(* IEC 61131-3 sources: MIRA/plc (part 4) *)

(* ---- Micro820_v4.2.2_Program.st ---- *)
PROGRAM Prog2
(* ================================================================ *)
(*  MIRA Conveyor Control -- Micro820 2080-LC20-20QBB               *)
(*  Version:  v4.2.2                                                *)
(*  Date:     2026-06-27                                            *)
(*  Author:   MIRA/Codex                                            *)
(*                                                                  *)
(*  v4.2.2 is a bench/demo logic update on top of v4.1.9. It adds   *)
(*  supervised SimLab discharge request handling for the garage      *)
(*  conveyor when used as bottling-line discharge_conveyor01. This  *)
(*  is not production-certified machinery control. The real         *)
(*  Micro820/GS10 bench still owns motion and safety authority.     *)
(*                                                                  *)
(*  Changelog vs v4.1.9:                                            *)
(*   0. FIX v4.2.2 -- remove the extra safety-ok global requirement. *)
(*      CCW build proved that variable was not in the v4.2.0 delta.  *)
(*      Use existing e_stop_active / estop_wiring_fault directly.    *)
(*   1. NEW -- simlab_discharge_request is request-only. It never   *)
(*      writes directly to the VFD, motor, contactor, or outputs.   *)
(*   2. NEW -- discharge_pending_acceptance requires a local human  *)
(*      acceptance rising edge from PBRun / _IO_EM_DI_04.           *)
(*   3. NEW -- discharge_accept_timer rejects pending requests      *)
(*      after 30 seconds if no local acceptance arrives.             *)
(*   4. NEW -- photoeye_clear_timer requires DI05/photoeye clear    *)
(*      for 30 seconds before the next accepted discharge can run.  *)
(*   5. NEW -- accepted discharge stops when photoeye_blocked goes  *)
(*      TRUE, or on E-stop, stop/selector-off, drive comm fault,    *)
(*      active fault, heartbeat loss, request drop, or shutdown.    *)
(*   6. NEW -- amber_led_flash now drives the bench amber lamp on   *)
(*      O-04 / _IO_EM_DO_04 while discharge acceptance is pending.  *)
(*      Do not reuse DO0/DO1/DO2/DO3.                               *)
(*                                                                  *)
(*  Still deliberately deferred beyond v4.2.2:                      *)
(*   - Removal of vfd_cmd_word := N assignments throughout the      *)
(*     state machine. The TODO calls for the motor_starter UDFB     *)
(*     in Prog4 to become the sole writer. Until Prog4 ships,       *)
(*     removing these writes here would leave nothing commanding    *)
(*     the drive. Two writers in one scan is bad, zero writers      *)
(*     is worse. Will rip them out atomically with the Prog4 add.   *)
(*   - mb_read_status -> mb_read_monitor rename. That's a CCW       *)
(*     IDE instance rename + cross-reference cleanup. Not safe to   *)
(*     do via ST edit alone; do it in CCW. Comments below use the   *)
(*     accurate name (mb_read_monitor) so the rename is obvious.    *)
(*   - Poll timer 500ms -> 50ms tuning. Cosmetic right now; first   *)
(*     prove comms work, then tune.                                 *)
(*                                                                  *)
(*  NEW VARIABLES to declare in CCW Controller Variables table      *)
(*  (PrjLibrary.accdb -- DO NOT add a VAR block here):              *)
(*                                                                  *)
(*    Name                          Type                  Init      *)
(*    ----                          ----                  ----      *)
(*    commissioning_mode            BOOL                  (none)    *)
(*    read_status_word_local_cfg    MSGMODBUSPARA_LOCAL   (none)    *)
(*    read_status_word_target_cfg   MSGMODBUSPARA_TARGET  (none)    *)
(*    read_status_word_data         MODBUSLOCADDR[1..1]   (none)    *)
(*    mb_read_status_word           MSG_MODBUS2           (none)    *)
(*    vfd_status_word               WORD                  (none)    *)
(*    vfd_running_bit               BOOL                  (none)    *)
(*    vfd_at_speed_bit              BOOL                  (none)    *)
(*    vfd_drive_fault               BOOL                  (none)    *)
(*    last_err_step                 INT                   (none)    *)
(*    last_err_at_uptime            DINT                  (none)    *)
(*    last_ok_at_uptime             DINT                  (none)    *)
(*    last_msg_error_id             INT                   (none)    *)
(*    read_err_count                DINT                  (none)    *)
(*    write_cmd_err_count           DINT                  (none)    *)
(*    write_freq_err_count          DINT                  (none)    *)
(*    fault_reset_err_count         DINT                  (none)    *)
(*    read_status_word_err_count    DINT                  (none)    *)
(*                                                                  *)
(*    v4.2.2 discharge acceptance variables:                        *)
(*    simlab_discharge_request       BOOL                  FALSE     *)
(*    simlab_discharge_heartbeat     BOOL                  FALSE     *)
(*    discharge_pending_acceptance   BOOL                  FALSE     *)
(*    discharge_accepted             BOOL                  FALSE     *)
(*    discharge_running              BOOL                  FALSE     *)
(*    discharge_complete             BOOL                  FALSE     *)
(*    discharge_rejected_or_faulted  BOOL                  FALSE     *)
(*    discharge_accept_timeout       BOOL                  FALSE     *)
(*    amber_led_flash                BOOL                  FALSE     *)
(*    green_start_pb                 BOOL                  FALSE     *)
(*    photoeye_blocked               BOOL                  FALSE     *)
(*    photoeye_clear_30s             BOOL                  FALSE     *)
(*    bench_permissive_ok            BOOL                  FALSE     *)
(*    local_stop_active              BOOL                  FALSE     *)
(*    remote_start_allowed           BOOL                  FALSE     *)
(*    manual_start_allowed           BOOL                  FALSE     *)
(*    green_start_rising             BOOL                  FALSE     *)
(*    prev_green_start_pb            BOOL                  FALSE     *)
(*    discharge_pending_was_active   BOOL                  FALSE     *)
(*    amber_blink_phase              BOOL                  FALSE     *)
(*    discharge_accept_timer         TON                   (none)    *)
(*    photoeye_clear_timer           TON                   (none)    *)
(*    amber_blink_timer              TON                   (none)    *)
(*                                                                  *)
(*  And expose them in MbSrvConf.xml so vfd_diag.py / live_monitor  *)
(*  / mira-bridge can read them over Modbus TCP. Suggested map:     *)
(*                                                                  *)
(*    HR400118 vfd_status_word                                      *)
(*    HR400119 last_err_step                                        *)
(*    HR400120 last_msg_error_id                                    *)
(*    HR400121 read_err_count        (low word of DINT)             *)
(*    HR400122 last_err_at_uptime    (low word of DINT)             *)
(*    HR400123 last_ok_at_uptime     (low word of DINT)             *)
(*    C23      vfd_running_bit                                      *)
(*    C24      vfd_at_speed_bit                                     *)
(*    C25      vfd_drive_fault                                      *)
(*    C26      commissioning_mode                                   *)
(*    C27      simlab_discharge_request       (write, bench only)   *)
(*    C28      simlab_discharge_heartbeat     (write, bench only)   *)
(*    C29      discharge_pending_acceptance                         *)
(*    C30      discharge_accepted                                   *)
(*    C31      discharge_running                                    *)
(*    C32      discharge_complete                                   *)
(*    C33      discharge_rejected_or_faulted                        *)
(*    C34      discharge_accept_timeout                             *)
(*    C35      amber_led_flash               (amber state readback) *)
(*    C36      green_start_pb                                       *)
(*    C37      photoeye_blocked                                      *)
(*    C38      photoeye_clear_30s                                   *)
(*    C39      bench_permissive_ok                                  *)
(*                                                                  *)
(*  Physical I/O (DO0-DO3 unchanged from v4.1.7/v4.1.8):            *)
(*    I-00 = SelectorFWD    O-00 = LightGreen (running)             *)
(*    I-01 = SelectorREV    O-01 = LightRed (fault/e-stop)          *)
(*    I-02 = EStopNC        O-02 = ContactorQ1 (safety)             *)
(*    I-03 = EStopNO        O-03 = PBRunLED (pushbutton light)      *)
(*    I-04 = PBRun                                                  *)
(*    I-05 = Photoeye / PE-101, confirm blocked polarity on bench    *)
(*                            O-04 = AmberLight (pending accept)    *)
(*                                                                  *)
(*  Only Prog2 may drive _IO_EM_DO_04. Before download, remove or    *)
(*  disable any legacy Prog1 rung that still drives DO4 as a          *)
(*  direction-indicator output.                                      *)
(*                                                                  *)
(*  VFD: AutomationDirect GS10 DURApulse                            *)
(*    RS-485 Modbus RTU, slave addr 1, 9600/8N2                     *)
(*    P09.00 = 1   (slave addr)                                     *)
(*    P09.01 = 96  (9600 baud)                                      *)
(*    P09.02 = 0   (warn + continue on comm loss -- confirmed)      *)
(*    P09.03 = 5   (5 sec timeout)                                  *)
(*    P09.04 = 13  (8N2 RTU)                                        *)
(*    P09.09 = 20  (response delay ms -- bump to 50 if CRC errs)    *)
(*    P00.21 = 2   (run source = RS-485)                            *)
(*                                                                  *)
(*    GS10 Register Map:                                            *)
(*      0x2000 (8192)  Control Command         (W FC06, bit field)  *)
(*      0x2001 (8193)  Frequency Setpoint      (W FC06, Hz x 10)    *)
(*      0x2002 (8194)  Fault Reset             (W FC06, write 2)    *)
(*      0x2101 (8449)  Status Word             (R FC03, bit field)  *)
(*      0x2103 (8451)  Output Frequency        (R FC03, Hz x 10)    *)
(*      0x2104 (8452)  Output Current          (R FC03, A x 10)     *)
(*      0x2105 (8453)  DC Bus Voltage          (R FC03, V)          *)
(*      0x2106 (8454)  Output Voltage          (R FC03, V)          *)
(*    Command bit-field: FWD+RUN=18  REV+RUN=20  STOP=1             *)
(* ================================================================ *)

  (* ================================================================ *)
  (* SECTION 1 -- E-STOP SUPERVISION (highest priority)               *)
  (* Existing v4.x E-stop state. Use the existing variables directly  *)
  (* so this package does not require a new safety-ok global.         *)
  (* ================================================================ *)
  IF (_IO_EM_DI_02 XOR _IO_EM_DI_03) THEN
    IF NOT _IO_EM_DI_02 AND _IO_EM_DI_03 THEN
      e_stop_active := TRUE;
    ELSE
      e_stop_active := FALSE;
    END_IF;
    estop_wiring_fault := FALSE;
  ELSE
    e_stop_active := TRUE;
    fault_alarm := TRUE;
    estop_wiring_fault := TRUE;
  END_IF;

  (* ================================================================ *)
  (* SECTION 2 -- OPERATOR STATION I/O MAPPING (unchanged)            *)
  (* ================================================================ *)
  dir_fwd := _IO_EM_DI_00 AND NOT _IO_EM_DI_01;
  dir_rev := NOT _IO_EM_DI_00 AND _IO_EM_DI_01;
  dir_off := NOT _IO_EM_DI_00 AND NOT _IO_EM_DI_01;
  dir_fault := _IO_EM_DI_00 AND _IO_EM_DI_01;

  sensor_1_active := _IO_EM_DI_05;
  sensor_2_active := _IO_EM_DI_06;

  green_start_pb := _IO_EM_DI_04;
  green_start_rising := green_start_pb AND NOT prev_green_start_pb;
  button_rising := green_start_rising;
  prev_green_start_pb := green_start_pb;
  prev_button := green_start_pb;

  photoeye_blocked := sensor_1_active;
  local_stop_active := dir_off;

  (* ================================================================ *)
  (* SECTION 3 -- SIMLAB DISCHARGE HUMAN ACCEPTANCE (bench/demo logic) *)
  (*                                                                  *)
  (* SimLab may request discharge, but the Micro820 remains control    *)
  (* authority. Remote request cannot start the conveyor directly.     *)
  (* Human acceptance requires a clean rising edge on PBRun / I-04.    *)
  (* This is bench/demo logic and not production-certified machinery   *)
  (* control.                                                         *)
  (* ================================================================ *)
  discharge_pending_was_active := discharge_pending_acceptance;

  photoeye_clear_timer(IN := NOT photoeye_blocked, PT := T#30s);
  photoeye_clear_30s := photoeye_clear_timer.Q;

  bench_permissive_ok :=
       NOT e_stop_active
   AND NOT estop_wiring_fault
   AND NOT local_stop_active
   AND NOT fault_alarm
   AND NOT dir_fault
   AND vfd_comm_ok
   AND NOT vfd_comm_err
   AND NOT vfd_drive_fault
   AND simlab_discharge_heartbeat
   AND NOT photoeye_blocked
   AND photoeye_clear_30s;

  manual_start_allowed :=
       green_start_rising
   AND (dir_fwd OR dir_rev)
   AND NOT simlab_discharge_request
   AND NOT discharge_pending_acceptance
   AND NOT discharge_accepted
   AND NOT discharge_running;

  remote_start_allowed :=
       discharge_accepted
   AND bench_permissive_ok
   AND (dir_fwd OR dir_rev)
   AND simlab_discharge_request
   AND simlab_discharge_heartbeat;

  discharge_accept_timer(IN := discharge_pending_acceptance, PT := T#30s);
  amber_blink_timer(IN := discharge_pending_acceptance AND NOT amber_blink_timer.Q, PT := T#500ms);

  IF NOT discharge_pending_acceptance THEN
    amber_blink_phase := FALSE;
  ELSIF amber_blink_timer.Q THEN
    amber_blink_phase := NOT amber_blink_phase;
  END_IF;
  amber_led_flash := discharge_pending_acceptance AND amber_blink_phase;

  IF NOT simlab_discharge_request THEN
    discharge_pending_acceptance := FALSE;
    discharge_accepted := FALSE;
    discharge_running := FALSE;
    discharge_complete := FALSE;
    discharge_rejected_or_faulted := FALSE;
    discharge_accept_timeout := FALSE;
  END_IF;

  IF simlab_discharge_request
     AND NOT discharge_pending_acceptance
     AND NOT discharge_accepted
     AND NOT discharge_running
     AND NOT discharge_complete
     AND NOT discharge_rejected_or_faulted
     AND NOT discharge_accept_timeout THEN
    discharge_pending_acceptance := TRUE;
  END_IF;

  IF discharge_pending_acceptance THEN
    motor_running := FALSE;
    conveyor_running := FALSE;
    vfd_cmd_word := 1;

    IF (NOT simlab_discharge_request) OR (NOT simlab_discharge_heartbeat) THEN
      discharge_pending_acceptance := FALSE;
      discharge_rejected_or_faulted := TRUE;
    ELSIF discharge_accept_timer.Q THEN
      discharge_pending_acceptance := FALSE;
      discharge_accept_timeout := TRUE;
      discharge_rejected_or_faulted := TRUE;
    ELSIF discharge_pending_was_active AND green_start_rising AND bench_permissive_ok THEN
      discharge_pending_acceptance := FALSE;
      discharge_accepted := TRUE;
    END_IF;
  END_IF;

  IF discharge_running AND photoeye_blocked THEN
    discharge_running := FALSE;
    discharge_accepted := FALSE;
    discharge_complete := TRUE;
  ELSIF discharge_running AND NOT bench_permissive_ok THEN
    discharge_running := FALSE;
    discharge_accepted := FALSE;
    discharge_rejected_or_faulted := TRUE;
  ELSIF discharge_running AND NOT simlab_discharge_request THEN
    discharge_running := FALSE;
    discharge_accepted := FALSE;
    discharge_rejected_or_faulted := TRUE;
  ELSIF discharge_running AND NOT simlab_discharge_heartbeat THEN
    discharge_running := FALSE;
    discharge_accepted := FALSE;
    discharge_rejected_or_faulted := TRUE;
  END_IF;

  (* ================================================================ *)
  (* SECTION 4 -- SAFETY CONTACTOR Q1 (O-02) (unchanged)              *)
  (* ================================================================ *)
  _IO_EM_DO_02 := NOT e_stop_active AND NOT estop_wiring_fault;

  (* ================================================================ *)
  (* SECTION 5 -- CONVEYOR STATE MACHINE                              *)
  (*                                                                  *)
  (* NOTE for v4.2.2: when Prog4 motor_starter UDFB exists, every     *)
  (* "vfd_cmd_word := N;" assignment in this section gets deleted,    *)
  (* and the UDFB becomes the sole writer of vfd_cmd_word. Until      *)
  (* then they stay, otherwise the drive gets no commands at all.    *)
  (* ================================================================ *)
  CASE conv_state OF

    0: (* IDLE *)
      motor_running := FALSE;
      conveyor_running := FALSE;
      motor_speed := 0;
      vfd_cmd_word := 1;

      IF fault_alarm OR e_stop_active OR dir_fault THEN
        conv_state := 4;
      ELSIF (manual_start_allowed OR remote_start_allowed) THEN
        conv_state := 1;
      END_IF;

    1: (* STARTING *)
      motor_running := TRUE;

      IF dir_fwd THEN
        vfd_cmd_word := 18;
      ELSIF dir_rev THEN
        vfd_cmd_word := 20;
      END_IF;

      IF e_stop_active OR fault_alarm OR dir_fault OR discharge_rejected_or_faulted THEN
        vfd_cmd_word := 1;
        conv_state := 4;
      ELSIF discharge_accepted AND NOT remote_start_allowed THEN
        vfd_cmd_word := 1;
        conv_state := 3;
      ELSIF start_timer.Q THEN
        conveyor_running := TRUE;
        conv_state := 2;
      END_IF;

    2: (* RUNNING *)
      motor_running := TRUE;
      conveyor_running := TRUE;

      IF dir_fwd THEN
        vfd_cmd_word := 18;
      ELSIF dir_rev THEN
        vfd_cmd_word := 20;
      END_IF;

      IF e_stop_active OR fault_alarm OR dir_fault OR discharge_rejected_or_faulted THEN
        vfd_cmd_word := 1;
        conv_state := 4;
      ELSIF dir_off OR discharge_complete OR (discharge_accepted AND NOT remote_start_allowed) THEN
        vfd_cmd_word := 1;
        conv_state := 3;
      END_IF;

      IF sensor_2_active AND NOT SensorEnd_Prev THEN
        item_count := item_count + 1;
      END_IF;
      SensorEnd_Prev := sensor_2_active;

      motor_speed := conveyor_speed_cmd;

    3: (* STOPPING *)
      motor_running := FALSE;
      vfd_cmd_word := 1;
      motor_speed := 0;

      IF e_stop_active OR fault_alarm THEN
        conv_state := 4;
      ELSIF stop_timer.Q THEN
        conveyor_running := FALSE;
        conv_state := 0;
      END_IF;

    4: (* FAULT *)
      motor_running := FALSE;
      conveyor_running := FALSE;
      vfd_cmd_word := 1;
      motor_speed := 0;

      IF e_stop_active THEN
        error_code := 6;
      ELSIF estop_wiring_fault THEN
        error_code := 7;
      ELSIF dir_fault THEN
        error_code := 8;
      ELSIF vfd_comm_err THEN
        error_code := 9;
      END_IF;

      IF button_rising AND NOT e_stop_active
         AND NOT estop_wiring_fault AND NOT dir_off THEN
        fault_alarm := FALSE;
        error_code := 0;
        vfd_fault_reset_pending := TRUE;
        conv_state := 0;
      END_IF;

  ELSE
    conv_state := 0;
  END_CASE;

  start_timer(IN := (conv_state = 1), PT := T#3000ms);
  stop_timer(IN := (conv_state = 3), PT := T#2000ms);

  IF discharge_accepted THEN
    discharge_running := motor_running AND ((conv_state = 1) OR (conv_state = 2));
  END_IF;

  (* ================================================================ *)
  (* SECTION 6 -- LED INDICATORS                                      *)
  (* ================================================================ *)
  IF ALL_LEDS_ON THEN
    _IO_EM_DO_00 := TRUE;
    _IO_EM_DO_01 := TRUE;
    _IO_EM_DO_03 := TRUE;
    _IO_EM_DO_04 := TRUE;
  ELSE
    _IO_EM_DO_00 := motor_running;
    _IO_EM_DO_01 := e_stop_active OR fault_alarm OR estop_wiring_fault
                     OR dir_fault OR (vfd_fault_code > 0);
    _IO_EM_DO_03 := motor_running;
    _IO_EM_DO_04 := amber_led_flash;
  END_IF;

  (* ================================================================ *)
  (* SECTION 7 -- VFD MODBUS RTU COMMUNICATION (v4.1.9 rebuild)       *)
  (*                                                                  *)
  (* 5-step poll cycle. Step skipped if vfd_poll_step lands on a       *)
  (* disabled step (commissioning_mode masks writes; fault_reset      *)
  (* only fires when pending).                                        *)
  (*                                                                  *)
  (*   Step 1: READ MONITOR  -- FC03 @ 0x2103, 4 regs (freq/cur/dc/v) *)
  (*   Step 2: WRITE CMD     -- FC06 @ 0x2000 (skipped if commission) *)
  (*   Step 3: WRITE FREQ    -- FC06 @ 0x2001 (skipped if commission) *)
  (*   Step 4: FAULT RESET   -- FC06 @ 0x2002 (only if pending)       *)
  (*   Step 5: READ STATUSW  -- FC03 @ 0x2101, 1 reg  (NEW v4.1.9)    *)
  (* ================================================================ *)

  (* --- Configure Modbus READ MONITOR (step 1, 0x2103, 4 regs) --- *)
  read_local_cfg.Channel := 2;
  read_local_cfg.TriggerType := 0;
  read_local_cfg.Cmd := 3;
  read_local_cfg.ElementCnt := 4;     (* v4.1.9: was 6, GS10 monitor block ends at 0x2106 *)
  read_target_cfg.Addr := 8451;       (* 0x2103 *)
  read_target_cfg.Node := 1;

  (* --- Configure Modbus WRITE COMMAND (step 2, 0x2000) --- *)
  write_cmd_local_cfg.Channel := 2;
  write_cmd_local_cfg.TriggerType := 0;
  write_cmd_local_cfg.Cmd := 6;
  write_cmd_local_cfg.ElementCnt := 1;
  write_cmd_target_cfg.Addr := 8192;   (* 0x2000 *)
  write_cmd_target_cfg.Node := 1;

  (* --- Configure Modbus WRITE FREQUENCY (step 3, 0x2001) --- *)
  write_freq_local_cfg.Channel := 2;
  write_freq_local_cfg.TriggerType := 0;
  write_freq_local_cfg.Cmd := 6;
  write_freq_local_cfg.ElementCnt := 1;
  write_freq_target_cfg.Addr := 8193;   (* 0x2001 *)
  write_freq_target_cfg.Node := 1;

  (* --- Configure Modbus FAULT RESET (step 4, 0x2002) --- *)
  fault_reset_local_cfg.Channel := 2;
  fault_reset_local_cfg.TriggerType := 0;
  fault_reset_local_cfg.Cmd := 6;
  fault_reset_local_cfg.ElementCnt := 1;
  fault_reset_target_cfg.Addr := 8194;   (* 0x2002 *)
  fault_reset_target_cfg.Node := 1;

  (* --- v4.1.9 NEW: Configure Modbus READ STATUS WORD (step 5, 0x2101) --- *)
  read_status_word_local_cfg.Channel := 2;
  read_status_word_local_cfg.TriggerType := 0;
  read_status_word_local_cfg.Cmd := 3;        (* FC03 *)
  read_status_word_local_cfg.ElementCnt := 1; (* single register *)
  read_status_word_target_cfg.Addr := 8449;   (* 0x2101 = Status Monitor 2 *)
  read_status_word_target_cfg.Node := 1;

  (* --- Compute VFD frequency setpoint --- *)
  vfd_freq_setpoint := conveyor_speed_cmd * 10;
  IF vfd_freq_setpoint = 0 AND motor_running THEN
    vfd_freq_setpoint := 300;
  END_IF;

  (* --- Load write data buffers via COP function blocks (unchanged from v4.1.8) --- *)
  fault_reset_cmd := 2;
  cop_cmd(Enable := TRUE, Src := vfd_cmd_word, SrcOffset := 0,
          Dest := write_cmd_data, DestOffset := 0, Length := 1, Swap := FALSE);
  cop_freq(Enable := TRUE, Src := vfd_freq_setpoint, SrcOffset := 0,
           Dest := write_freq_data, DestOffset := 0, Length := 1, Swap := FALSE);
  cop_reset(Enable := TRUE, Src := fault_reset_cmd, SrcOffset := 0,
            Dest := fault_reset_data, DestOffset := 0, Length := 1, Swap := FALSE);

  (* --- Poll timer: 500ms between each MSG step (tune only after comms proof) --- *)
  vfd_poll_timer(IN := NOT vfd_poll_active, PT := T#500ms);

  IF vfd_poll_timer.Q AND NOT vfd_poll_active THEN
    vfd_poll_active := TRUE;
    vfd_msg_done := FALSE;
    vfd_poll_step := vfd_poll_step + 1;
    IF vfd_poll_step > 5 THEN
      vfd_poll_step := 1;
    END_IF;

    (* Skip fault reset step unless a reset is pending *)
    IF vfd_poll_step = 4 AND NOT vfd_fault_reset_pending THEN
      vfd_poll_step := 5;
    END_IF;

    (* v4.1.9 NEW: commissioning_mode masks writes -- only steps 1 and 5 *)
    (* (the two reads) fire. Lets us prove bidirectional comms without  *)
    (* commanding the drive. Drop back to step 1 on every other step.   *)
    IF commissioning_mode AND (vfd_poll_step = 2 OR vfd_poll_step = 3
                                OR vfd_poll_step = 4) THEN
      vfd_poll_step := 5;
    END_IF;
  END_IF;

  (* --- Call all five MSG blocks once per scan, only one fires --- *)
  (* mb_read_status is the OLD name for what should be mb_read_monitor.  *)
  (* Rename the FB instance in CCW for v4.2.2. Keeping the old name      *)
  (* here so this file compiles without an IDE-side rename.              *)
  mb_read_status(IN := (vfd_poll_step = 1) AND vfd_poll_active,
                 LocalCfg := read_local_cfg,
                 TargetCfg := read_target_cfg,
                 LocalAddr := read_data);

  mb_write_cmd(IN := (vfd_poll_step = 2) AND vfd_poll_active,
               LocalCfg := write_cmd_local_cfg,
               TargetCfg := write_cmd_target_cfg,
               LocalAddr := write_cmd_data);

  mb_write_freq(IN := (vfd_poll_step = 3) AND vfd_poll_active,
                LocalCfg := write_freq_local_cfg,
                TargetCfg := write_freq_target_cfg,
                LocalAddr := write_freq_data);

  mb_fault_reset(IN := (vfd_poll_step = 4) AND vfd_poll_active,
                 LocalCfg := fault_reset_local_cfg,
                 TargetCfg := fault_reset_target_cfg,
                 LocalAddr := fault_reset_data);

  mb_read_status_word(IN := (vfd_poll_step = 5) AND vfd_poll_active,
                      LocalCfg := read_status_word_local_cfg,
                      TargetCfg := read_status_word_target_cfg,
                      LocalAddr := read_status_word_data);

  (* --- Check MSG results (v4.1.9: per-step counters + last_err_step) --- *)
  IF vfd_poll_active AND NOT vfd_msg_done THEN
    CASE vfd_poll_step OF
      1: (* READ MONITOR *)
        IF mb_read_status.Q THEN
          vfd_frequency := read_data(1);
          vfd_current   := read_data(2);
          vfd_dc_bus    := read_data(3);
          vfd_voltage   := read_data(4);
          vfd_comm_ok   := TRUE;
          vfd_comm_err  := FALSE;
          last_ok_at_uptime := uptime_seconds;
          vfd_msg_done := TRUE;
          vfd_poll_active := FALSE;
        END_IF;
        IF mb_read_status.Error THEN
          vfd_comm_ok := FALSE;
          vfd_comm_err := TRUE;
          read_err_count := read_err_count + 1;
          last_err_step := 1;
          last_err_at_uptime := uptime_seconds;
          last_msg_error_id := mb_read_status.ErrorID;
          vfd_msg_done := TRUE;
          vfd_poll_active := FALSE;
        END_IF;

      2: (* WRITE COMMAND *)
        IF mb_write_cmd.Q THEN
          last_ok_at_uptime := uptime_seconds;
          vfd_msg_done := TRUE;
          vfd_poll_active := FALSE;
        END_IF;
        IF mb_write_cmd.Error THEN
          vfd_comm_err := TRUE;
          write_cmd_err_count := write_cmd_err_count + 1;
          last_err_step := 2;
          last_err_at_uptime := uptime_seconds;
          last_msg_error_id := mb_write_cmd.ErrorID;
          vfd_msg_done := TRUE;
          vfd_poll_active := FALSE;
        END_IF;

      3: (* WRITE FREQUENCY *)
        IF mb_write_freq.Q THEN
          last_ok_at_uptime := uptime_seconds;
          vfd_msg_done := TRUE;
          vfd_poll_active := FALSE;
        END_IF;
        IF mb_write_freq.Error THEN
          vfd_comm_err := TRUE;
          write_freq_err_count := write_freq_err_count + 1;
          last_err_step := 3;
          last_err_at_uptime := uptime_seconds;
          last_msg_error_id := mb_write_freq.ErrorID;
          vfd_msg_done := TRUE;
          vfd_poll_active := FALSE;
        END_IF;

      4: (* FAULT RESET *)
        IF mb_fault_reset.Q THEN
          vfd_fault_reset_pending := FALSE;
          last_ok_at_uptime := uptime_seconds;
          vfd_msg_done := TRUE;
          vfd_poll_active := FALSE;
        END_IF;
        IF mb_fault_reset.Error THEN
          vfd_comm_err := TRUE;
          fault_reset_err_count := fault_reset_err_count + 1;
          last_err_step := 4;
          last_err_at_uptime := uptime_seconds;
          last_msg_error_id := mb_fault_reset.ErrorID;
          vfd_msg_done := TRUE;
          vfd_poll_active := FALSE;
        END_IF;

      5: (* READ STATUS WORD -- v4.1.9 NEW *)
        IF mb_read_status_word.Q THEN
          vfd_status_word := read_status_word_data(1);
          (* GS10 0x2101 bit map (per AutomationDirect GS10 user manual): *)
          (*   bit 0..1  = 00 stop / 01 decel / 10 standby / 11 running   *)
          (*   bit 2     = JOG cmd                                        *)
          (*   bit 3..4  = 00 stop / 01 decel / 10 standby / 11 running   *)
          (*               (direction status)                             *)
          (*   bit 8     = master freq controlled by comm                 *)
          (*   bit 9     = master freq controlled by analog               *)
          (*   bit 11    = operation cmd controlled by comm               *)
          (*   bit 12    = parameter is locked                            *)
          (*   bit 13    = drive is in fault                              *)
          vfd_running_bit := (vfd_status_word AND 16#0003) = 16#0003;
          vfd_at_speed_bit := (vfd_status_word AND 16#000C) = 16#000C;
          vfd_drive_fault := (vfd_status_word AND 16#2000) <> 0;
          vfd_comm_ok := TRUE;
          vfd_comm_err := FALSE;
          last_ok_at_uptime := uptime_seconds;
          vfd_msg_done := TRUE;
          vfd_poll_active := FALSE;
        END_IF;
        IF mb_read_status_word.Error THEN
          vfd_comm_ok := FALSE;
          vfd_comm_err := TRUE;
          read_status_word_err_count := read_status_word_err_count + 1;
          last_err_step := 5;
          last_err_at_uptime := uptime_seconds;
          last_msg_error_id := mb_read_status_word.ErrorID;
          vfd_msg_done := TRUE;
          vfd_poll_active := FALSE;
        END_IF;

    ELSE
      vfd_poll_step := 1;
      vfd_poll_active := FALSE;
    END_CASE;
  END_IF;

  (* --- VFD comm watchdog (unchanged) --- *)
  vfd_err_timer(IN := vfd_comm_err, PT := T#5000ms);
  IF vfd_err_timer.Q THEN
    fault_alarm := TRUE;
    error_code := 9;
  END_IF;

  (* ================================================================ *)
  (* SECTION 8 -- DIAGNOSTICS (inherited from v4.1.9)                *)
  (* ================================================================ *)
  heartbeat := NOT heartbeat;
  cycle_count := cycle_count + 1;
  uptime_timer(IN := NOT uptime_timer.Q, PT := T#1000ms);
  IF uptime_timer.Q THEN
    uptime_seconds := uptime_seconds + 1;
  END_IF;
  system_ready := NOT fault_alarm AND NOT e_stop_active AND (conv_state = 2);
  motor_stopped := NOT motor_running;
  conveyor_speed := conveyor_speed_cmd;

END_PROGRAM

(* ---- Micro820_v5.1.0_Program.st ---- *)
PROGRAM Prog2
(* ================================================================ *)
(*  MIRA Conveyor Control -- Micro820 2080-LC20-20QBB               *)
(*  Version:  v5.1.0  (Trends V2 -- full GS10 monitoring)           *)
(*  Date:     2026-06-12                                            *)
(*  Author:   MIRA/Claude                                           *)
(*                                                                  *)
(*  Changelog:                                                      *)
(*  v5.1.0 - Trends V2 (docs/plans/2026-06-12-trends-v2-full-vfd-   *)
(*           monitoring.md). Based on DEPLOYED v5.0.0 (Prog2.stf),  *)
(*           NOT the stale Micro820_v4.1.9_Program.st.              *)
(*           1. Step-1 read widened: 0x2103 x6 -> 0x2100 x7. One    *)
(*              FC03 now covers the whole documented monitor block: *)
(*              Status Monitor 1 (warn|error bytes), Status         *)
(*              Monitor 2 (status bits), freq command, output       *)
(*              freq/current/DC bus/voltage. read_data indices      *)
(*              shift by +3 -- decode below re-indexed.             *)
(*           2. SM1 byte split -> vfd_fault_code (low byte, was     *)
(*              never written before -- the red-light term          *)
(*              vfd_fault_code > 0 now actually fires) and NEW      *)
(*              vfd_warn_code (high byte).                          *)
(*           3. NEW vfd_last_fault latch: holds the last nonzero    *)
(*              fault code; survives the drive's own fault reset.   *)
(*              Cleared ONLY by operator coil last_fault_clear.     *)
(*           4. NEW steps 5/6: FC03 0x210B x2 (torque %x10, motor   *)
(*              rpm) and FC03 0x210F x1 (power kW x1000).           *)
(*              Separate reads -- 0x210D/0x210E are reserved; do    *)
(*              not span them in one transaction.                   *)
(*           5. Poll cycle 4 -> 6 steps; fault-reset skip now goes  *)
(*              4 -> 5 (was 4 -> 1) so the new reads still fire.    *)
(*  v5.0.0 - Clean rebuild from v4.1.9. Per-step MSG timeout so     *)
(*           poll never hangs if serial driver is not loaded.       *)
(*           Channel 0 = built-in RS-485 (confirmed Rockwell docs). *)
(*                                                                  *)
(*  NOTE: All variables declared in CCW Controller Variables table  *)
(*        (PrjLibrary.accdb). Do NOT add a VAR block here.          *)
(*        NEW variables for v5.1.0: see                             *)
(*        plc/CCW_VARIABLES_v5.1.0_DELTA.md                         *)
(*                                                                  *)
(*  Physical I/O:                                                   *)
(*    I-00 = SelectorFWD    O-00 = LightGreen (running)             *)
(*    I-01 = SelectorREV    O-01 = LightRed (fault/e-stop)          *)
(*    I-02 = EStopNC        O-02 = ContactorQ1 (safety)             *)
(*    I-03 = EStopNO        O-03 = PBRunLED (pushbutton light)      *)
(*    I-04 = PBRun                                                  *)
(*                                                                  *)
(*  VFD: AutomationDirect GS10 DURApulse                            *)
(*    RS-485 Modbus RTU, slave addr 1, 9600/8N2                     *)
(*    Command register:  0x2000 (8192) -- bit field                 *)
(*    Freq setpoint reg: 0x2001 (8193) -- Hz x 10                   *)
(*    Fault reset reg:   0x2002 (8194) -- write 2 to reset          *)
(*    Monitor block:     0x2100 (8448) x7 -- SM1, SM2, freq cmd,    *)
(*                       out freq, current, DC bus, out voltage     *)
(*    Load block:        0x210B (8459) x2 -- torque %x10, rpm       *)
(*    Power:             0x210F (8463) x1 -- kW x1000               *)
(*    FWD+RUN=18  REV+RUN=20  STOP=1                               *)
(*                                                                  *)
(*    GS10 0x2101 Status Monitor 2 bits (UM 1st Ed Rev B p4-196):   *)
(*      bits 1-0: 00 stop / 01 decel / 10 standby / 11 operating    *)
(*      bit  2:   JOG command                                       *)
(*      bits 4-3: 00 FWD / 01 REV->FWD / 10 FWD->REV / 11 REV       *)
(*      bit  8:   master freq from comms                            *)
(*      bit  9:   master freq from analog/terminal                  *)
(*      bit 10:   operation command from comms                      *)
(*      bit 11:   parameters locked                                 *)
(*      bit 12:   keypad copy enabled                               *)
(*      bits 15-13: reserved                                        *)
(*      (The v4.1.9 comment claimed bit 13 = drive fault. The       *)
(*       manual has no such bit -- fault truth is SM1 low byte.)    *)
(* ================================================================ *)

  (* ================================================================ *)
  (* SECTION 1 -- E-STOP SUPERVISION (highest priority)               *)
  (*   I-02 (EStopNC) = NC contact (healthy = 1, pressed = 0)        *)
  (*   I-03 (EStopNO) = NO contact (healthy = 0, pressed = 1)        *)
  (*   Dual-channel: I-02 XOR I-03 must be TRUE                      *)
  (* ================================================================ *)
  IF (_IO_EM_DI_02 XOR _IO_EM_DI_03) THEN
    IF NOT _IO_EM_DI_02 AND _IO_EM_DI_03 THEN
      e_stop_active := TRUE;
    ELSE
      e_stop_active := FALSE;
    END_IF;
    estop_wiring_fault := FALSE;
  ELSE
    e_stop_active := TRUE;
    fault_alarm := TRUE;
    estop_wiring_fault := TRUE;
  END_IF;

  (* ================================================================ *)
  (* SECTION 2 -- OPERATOR STATION I/O MAPPING                       *)
  (* ================================================================ *)
  dir_fwd := _IO_EM_DI_00 AND NOT _IO_EM_DI_01;
  dir_rev := NOT _IO_EM_DI_00 AND _IO_EM_DI_01;
  dir_off := NOT _IO_EM_DI_00 AND NOT _IO_EM_DI_01;
  dir_fault := _IO_EM_DI_00 AND _IO_EM_DI_01;

  sensor_1_active := _IO_EM_DI_05;
  sensor_2_active := _IO_EM_DI_06;

  button_rising := _IO_EM_DI_04 AND NOT prev_button;
  prev_button := _IO_EM_DI_04;

  (* ================================================================ *)
  (* SECTION 3 -- SAFETY CONTACTOR Q1 (O-02)                         *)
  (* ================================================================ *)
  _IO_EM_DO_02 := NOT e_stop_active AND NOT estop_wiring_fault;

  (* ================================================================ *)
  (* SECTION 4 -- CONVEYOR STATE MACHINE                              *)
  (*   States: 0=IDLE, 1=STARTING, 2=RUNNING, 3=STOPPING, 4=FAULT    *)
  (* ================================================================ *)
  CASE conv_state OF

    0: (* IDLE *)
      motor_running := FALSE;
      conveyor_running := FALSE;
      motor_speed := 0;
      vfd_cmd_word := 1;

      IF fault_alarm OR e_stop_active OR dir_fault THEN
        conv_state := 4;
      ELSIF button_rising AND (dir_fwd OR dir_rev) THEN
        conv_state := 1;
      END_IF;

    1: (* STARTING *)
      motor_running := TRUE;
      IF dir_fwd THEN
        vfd_cmd_word := 18;
      ELSIF dir_rev THEN
        vfd_cmd_word := 20;
      END_IF;

      IF e_stop_active OR fault_alarm OR dir_fault THEN
        vfd_cmd_word := 1;
        conv_state := 4;
      ELSIF start_timer.Q THEN
        conveyor_running := TRUE;
        conv_state := 2;
      END_IF;

    2: (* RUNNING *)
      motor_running := TRUE;
      conveyor_running := TRUE;
      IF dir_fwd THEN
        vfd_cmd_word := 18;
      ELSIF dir_rev THEN
        vfd_cmd_word := 20;
      END_IF;

      IF e_stop_active OR fault_alarm OR dir_fault THEN
        vfd_cmd_word := 1;
        conv_state := 4;
      ELSIF dir_off THEN
        vfd_cmd_word := 1;
        conv_state := 3;
      END_IF;

      IF sensor_2_active AND NOT SensorEnd_Prev THEN
        item_count := item_count + 1;
      END_IF;
      SensorEnd_Prev := sensor_2_active;
      motor_speed := conveyor_speed_cmd;

    3: (* STOPPING *)
      motor_running := FALSE;
      vfd_cmd_word := 1;
      motor_speed := 0;

      IF e_stop_active OR fault_alarm THEN
        conv_state := 4;
      ELSIF stop_timer.Q THEN
        conveyor_running := FALSE;
        conv_state := 0;
      END_IF;

    4: (* FAULT *)
      motor_running := FALSE;
      conveyor_running := FALSE;
      vfd_cmd_word := 1;
      motor_speed := 0;

      IF e_stop_active THEN
        error_code := 6;
      ELSIF estop_wiring_fault THEN
        error_code := 7;
      ELSIF dir_fault THEN
        error_code := 8;
      ELSIF vfd_comm_err THEN
        error_code := 9;
      END_IF;

      IF button_rising AND NOT e_stop_active
         AND NOT estop_wiring_fault AND NOT dir_off THEN
        fault_alarm := FALSE;
        error_code := 0;
        vfd_fault_reset_pending := TRUE;
        conv_state := 0;
      END_IF;

  ELSE
    conv_state := 0;
  END_CASE;

  start_timer(IN := (conv_state = 1), PT := T#3000ms);
  stop_timer(IN := (conv_state = 3), PT := T#2000ms);

  (* ================================================================ *)
  (* SECTION 5 -- LED INDICATORS                                      *)
  (* ================================================================ *)
  IF ALL_LEDS_ON THEN
    _IO_EM_DO_00 := TRUE;
    _IO_EM_DO_01 := TRUE;
    _IO_EM_DO_03 := TRUE;
  ELSE
    _IO_EM_DO_00 := motor_running;
    _IO_EM_DO_01 := e_stop_active OR fault_alarm OR estop_wiring_fault
                     OR dir_fault OR (vfd_fault_code > 0);
    _IO_EM_DO_03 := motor_running;
  END_IF;

  (* ================================================================ *)
  (* SECTION 6 -- VFD MODBUS RTU COMMUNICATION (v5.1.0 Trends V2)    *)
  (*   Channel 0 = built-in RS-485 serial port on 2080-LC20-20QBB    *)
  (*   GS10 DURApulse at slave address 1, 9600 baud, 8N2             *)
  (*                                                                  *)
  (*   Six MSG steps cycle:                                           *)
  (*     1: READ MONITOR -- FC03 0x2100 x7 (SM1/SM2/freq cmd/out     *)
  (*        freq/current/DC bus/out voltage)                          *)
  (*     2: WRITE CMD    -- FC06 0x2000                               *)
  (*     3: WRITE FREQ   -- FC06 0x2001                               *)
  (*     4: FAULT RESET  -- FC06 0x2002 (only when pending,           *)
  (*        otherwise skip straight to 5)                             *)
  (*     5: READ LOAD    -- FC03 0x210B x2 (torque, rpm)              *)
  (*     6: READ POWER   -- FC03 0x210F x1 (kW x1000)                 *)
  (*                                                                  *)
  (*   v5.0: msg_step_timer -- 2s timeout per step. If neither Q nor  *)
  (*   Error fires within 2s, the step is force-completed with an     *)
  (*   error. Prevents silent hangs when the serial driver is not     *)
  (*   loaded (ErrorID=255).                                          *)
  (* ================================================================ *)

  (* --- Configure Modbus READ MONITOR parameters (v5.1.0: 0x2100 x7) --- *)
  read_local_cfg.Channel := 0;
  read_local_cfg.TriggerType := 0;
  read_local_cfg.Cmd := 3;
  read_local_cfg.ElementCnt := 7;
  read_target_cfg.Addr := 8448;
  read_target_cfg.Node := 1;

  (* --- Configure Modbus WRITE COMMAND parameters --- *)
  write_cmd_local_cfg.Channel := 0;
  write_cmd_local_cfg.TriggerType := 0;
  write_cmd_local_cfg.Cmd := 6;
  write_cmd_local_cfg.ElementCnt := 1;
  write_cmd_target_cfg.Addr := 8192;
  write_cmd_target_cfg.Node := 1;

  (* --- Configure Modbus WRITE FREQUENCY parameters --- *)
  write_freq_local_cfg.Channel := 0;
  write_freq_local_cfg.TriggerType := 0;
  write_freq_local_cfg.Cmd := 6;
  write_freq_local_cfg.ElementCnt := 1;
  write_freq_target_cfg.Addr := 8193;
  write_freq_target_cfg.Node := 1;

  (* --- Configure Modbus FAULT RESET parameters --- *)
  fault_reset_local_cfg.Channel := 0;
  fault_reset_local_cfg.TriggerType := 0;
  fault_reset_local_cfg.Cmd := 6;
  fault_reset_local_cfg.ElementCnt := 1;
  fault_reset_target_cfg.Addr := 8194;
  fault_reset_target_cfg.Node := 1;

  (* --- v5.1.0 NEW: Configure Modbus READ LOAD parameters (0x210B x2) --- *)
  read_load_local_cfg.Channel := 0;
  read_load_local_cfg.TriggerType := 0;
  read_load_local_cfg.Cmd := 3;
  read_load_local_cfg.ElementCnt := 2;
  read_load_target_cfg.Addr := 8459;
  read_load_target_cfg.Node := 1;

  (* --- v5.1.0 NEW: Configure Modbus READ POWER parameters (0x210F x1) --- *)
  read_power_local_cfg.Channel := 0;
  read_power_local_cfg.TriggerType := 0;
  read_power_local_cfg.Cmd := 3;
  read_power_local_cfg.ElementCnt := 1;
  read_power_target_cfg.Addr := 8463;
  read_power_target_cfg.Node := 1;

  (* --- Compute VFD frequency setpoint --- *)
  vfd_freq_setpoint := conveyor_speed_cmd * 10;
  IF vfd_freq_setpoint = 0 AND motor_running THEN
    vfd_freq_setpoint := 300;
  END_IF;

  (* --- Load write data buffers via COP --- *)
  fault_reset_cmd := 2;
  cop_cmd(Enable := TRUE, Src := vfd_cmd_word, SrcOffset := 0,
          Dest := write_cmd_data, DestOffset := 0, Length := 1, Swap := FALSE);
  cop_freq(Enable := TRUE, Src := vfd_freq_setpoint, SrcOffset := 0,
           Dest := write_freq_data, DestOffset := 0, Length := 1, Swap := FALSE);
  cop_reset(Enable := TRUE, Src := fault_reset_cmd, SrcOffset := 0,
            Dest := fault_reset_data, DestOffset := 0, Length := 1, Swap := FALSE);

  (* --- Poll timer: 500ms between each MSG step --- *)
  vfd_poll_timer(IN := NOT vfd_poll_active, PT := T#500ms);

  IF vfd_poll_timer.Q AND NOT vfd_poll_active THEN
    vfd_poll_active := TRUE;
    vfd_msg_done := FALSE;
    vfd_poll_step := vfd_poll_step + 1;
    IF vfd_poll_step > 6 THEN
      vfd_poll_step := 1;
    END_IF;
    (* v5.1.0: skip fault reset to the NEW read steps, not back to 1 *)
    IF vfd_poll_step = 4 AND NOT vfd_fault_reset_pending THEN
      vfd_poll_step := 5;
    END_IF;
  END_IF;

  (* --- Per-step timeout: 2s max per MSG transaction --- *)
  (* v5.0: catches silent failures when serial driver not loaded *)
  msg_step_timer(IN := vfd_poll_active AND NOT vfd_msg_done, PT := T#2000ms);
  IF msg_step_timer.Q THEN
    vfd_comm_ok := FALSE;
    vfd_comm_err := TRUE;
    vfd_msg_done := TRUE;
    vfd_poll_active := FALSE;
  END_IF;

  (* --- Call all six MSG blocks once per scan --- *)
  mb_read_status(IN := (vfd_poll_step = 1) AND vfd_poll_active,
                 LocalCfg := read_local_cfg,
                 TargetCfg := read_target_cfg,
                 LocalAddr := read_data);

  mb_write_cmd(IN := (vfd_poll_step = 2) AND vfd_poll_active,
               LocalCfg := write_cmd_local_cfg,
               TargetCfg := write_cmd_target_cfg,
               LocalAddr := write_cmd_data);

  mb_write_freq(IN := (vfd_poll_step = 3) AND vfd_poll_active,
                LocalCfg := write_freq_local_cfg,
                TargetCfg := write_freq_target_cfg,
                LocalAddr := write_freq_data);

  mb_fault_reset(IN := (vfd_poll_step = 4) AND vfd_poll_active,
                 LocalCfg := fault_reset_local_cfg,
                 TargetCfg := fault_reset_target_cfg,
                 LocalAddr := fault_reset_data);

  mb_read_load(IN := (vfd_poll_step = 5) AND vfd_poll_active,
               LocalCfg := read_load_local_cfg,
               TargetCfg := read_load_target_cfg,
               LocalAddr := read_load_data);

  mb_read_power(IN := (vfd_poll_step = 6) AND vfd_poll_active,
                LocalCfg := read_power_local_cfg,
                TargetCfg := read_power_target_cfg,
                LocalAddr := read_power_data);

  (* --- Check MSG results --- *)
  IF vfd_poll_active AND NOT vfd_msg_done THEN
    CASE vfd_poll_step OF
      1: (* READ MONITOR -- v5.1.0 re-indexed: block starts at 0x2100 *)
        IF mb_read_status.Q THEN
          (* SM1 0x2100: high byte = warning code, low byte = fault code *)
          vfd_fault_code := read_data(1) AND 16#00FF;
          vfd_warn_code := SHR(read_data(1), 8);
          (* SM2 0x2101: status bits -- decoded downstream (trend viewer) *)
          vfd_status_word := read_data(2);
          (* 0x2102: commanded frequency (same scale as output freq) *)
          vfd_freq_cmd := read_data(3);
          vfd_frequency := read_data(4);
          vfd_current := read_data(5);
          vfd_dc_bus := read_data(6);
          vfd_voltage := read_data(7);

          (* v5.1.0: latch the trip cause. The drive zeroes SM1 low    *)
          (* byte on its own fault reset; this latch keeps the last    *)
          (* nonzero code until an operator deliberately clears it     *)
          (* via the last_fault_clear coil (C24).                      *)
          IF vfd_fault_code > 0 THEN
            vfd_last_fault := vfd_fault_code;
          END_IF;

          vfd_comm_ok := TRUE;
          vfd_comm_err := FALSE;
          vfd_msg_done := TRUE;
          vfd_poll_active := FALSE;
        END_IF;
        IF mb_read_status.Error THEN
          vfd_comm_ok := FALSE;
          vfd_comm_err := TRUE;
          vfd_msg_done := TRUE;
          vfd_poll_active := FALSE;
        END_IF;

      2:
        IF mb_write_cmd.Q OR mb_write_cmd.Error THEN
          IF mb_write_cmd.Error THEN
            vfd_comm_err := TRUE;
          END_IF;
          vfd_msg_done := TRUE;
          vfd_poll_active := FALSE;
        END_IF;

      3:
        IF mb_write_freq.Q OR mb_write_freq.Error THEN
          IF mb_write_freq.Error THEN
            vfd_comm_err := TRUE;
          END_IF;
          vfd_msg_done := TRUE;
          vfd_poll_active := FALSE;
        END_IF;

      4:
        IF mb_fault_reset.Q OR mb_fault_reset.Error THEN
          vfd_fault_reset_pending := FALSE;
          vfd_msg_done := TRUE;
          vfd_poll_active := FALSE;
        END_IF;

      5: (* READ LOAD -- v5.1.0 NEW: torque % x10, motor speed rpm *)
        IF mb_read_load.Q THEN
          vfd_torque := read_load_data(1);
          vfd_motor_rpm := read_load_data(2);
          vfd_comm_ok := TRUE;
          vfd_comm_err := FALSE;
          vfd_msg_done := TRUE;
          vfd_poll_active := FALSE;
        END_IF;
        IF mb_read_load.Error THEN
          vfd_comm_err := TRUE;
          vfd_msg_done := TRUE;
          vfd_poll_active := FALSE;
        END_IF;

      6: (* READ POWER -- v5.1.0 NEW: kW x1000 *)
        IF mb_read_power.Q THEN
          vfd_power := read_power_data(1);
          vfd_comm_ok := TRUE;
          vfd_comm_err := FALSE;
          vfd_msg_done := TRUE;
          vfd_poll_active := FALSE;
        END_IF;
        IF mb_read_power.Error THEN
          vfd_comm_err := TRUE;
          vfd_msg_done := TRUE;
          vfd_poll_active := FALSE;
        END_IF;

    ELSE
      vfd_poll_step := 1;
      vfd_poll_active := FALSE;
    END_CASE;
  END_IF;

  (* --- v5.1.0: operator clear for the last-fault latch (coil C24) --- *)
  IF last_fault_clear THEN
    vfd_last_fault := 16#0000;
    last_fault_clear := FALSE;
  END_IF;

  (* --- VFD comm watchdog: 5s of errors latches fault --- *)
  vfd_err_timer(IN := vfd_comm_err, PT := T#5000ms);
  IF vfd_err_timer.Q THEN
    fault_alarm := TRUE;
    error_code := 9;
  END_IF;

  (* ================================================================ *)
  (* SECTION 7 -- DIAGNOSTICS                                        *)
  (* ================================================================ *)
  heartbeat := NOT heartbeat;
  cycle_count := cycle_count + 1;
  uptime_timer(IN := NOT uptime_timer.Q, PT := T#1000ms);
  IF uptime_timer.Q THEN
    uptime_seconds := uptime_seconds + 1;
  END_IF;
  system_ready := NOT fault_alarm AND NOT e_stop_active AND (conv_state = 2);
  motor_stopped := NOT motor_running;
  conveyor_speed := conveyor_speed_cmd;

END_PROGRAM

(* ---- Prog1_ConvSimple_v2.2.st ---- *)
PROGRAM Prog1
#info= QLD
BOF

(**)

SOR  [0,1] (**) (**)  XIC  [1,0] (*_IO_EM_DI_02*) (*estop_nc*)  XIO  [2,0] (*_IO_EM_DI_03*) (*estop_no*)  OTE  [3,0] (*e_stop_ok*) (**)
EOR [4,0]

(**)

SOR  [0,3] (**) (**)  XIO  [1,0] (*_IO_EM_DI_02*) (*estop_nc*)  XIC  [2,0] (*_IO_EM_DI_03*) (*estop_no*)  OTE  [3,0] (*e_stop_active*) (**)
EOR [4,0]

(**)

SOR  [0,5] (**) (**)
 BST  XIC  [1,0] (*_IO_EM_DI_02*) (*estop_nc*)  XIC  [2,0] (*_IO_EM_DI_03*) (*estop_no*)
   NXB  XIO  [1,1] (*_IO_EM_DI_02*) (*estop_nc*)  XIO  [2,1] (*_IO_EM_DI_03*) (*estop_no*)
 BND
  OTE  [3,0] (*estop_wiring_fault*) (**)
EOR [4,0]

(**)

SOR  [0,8] (**) (**)  XIC  [1,0] (*e_stop_ok*) (**)
 BST  XIC  [2,0] (*_IO_EM_DI_04*) (*pb_start*)
   NXB  XIC  [2,1] (*_IO_EM_DO_02*) (**)
 BND
  OTE  [3,0] (*_IO_EM_DO_02*) (**)
EOR [4,0]

(**)

SOR  [0,11] (**) (**)  XIC  [1,0] (*amber_led_flash*) (*pending_accept*)  OTE  [2,0] (*_IO_EM_DO_04*) (*amber_light*)
EOR [4,0]

(**)

SOR  [0,13] (**) (**)  XIC  [1,0] (*_IO_EM_DI_01*) (*dir_rev_sw*)  XIO  [2,0] (*_IO_EM_DI_00*) (*dir_fwd_sw*)  OTE  [3,0] (*_IO_EM_DO_05*) (**)
EOR [4,0]

(**)

SOR  [0,15] (**) (**)  XIC  [1,0] (*_IO_EM_DO_02*) (**)  OTE  [2,0] (*_IO_EM_DO_00*) (*green_light*)
EOR [3,0]

(**)

SOR  [0,17] (**) (**)  XIO  [1,0] (*e_stop_ok*) (**)  OTE  [2,0] (*_IO_EM_DO_01*) (*red_light*)
EOR [3,0]
EOF
#end_info
END_PROGRAM

(* ---- Prog1_ConvSimple_v2.4.st ---- *)
PROGRAM Prog1
#info= QLD
BOF

(**)

SOR  [0,1] (**) (**)  XIC  [1,0] (*_IO_EM_DI_02*) (*estop_nc*)  XIO  [2,0] (*_IO_EM_DI_03*) (*estop_no*)  OTE  [3,0] (*e_stop_ok*) (**)
EOR [4,0]

(**)

SOR  [0,3] (**) (**)  XIO  [1,0] (*_IO_EM_DI_02*) (*estop_nc*)  XIC  [2,0] (*_IO_EM_DI_03*) (*estop_no*)  OTE  [3,0] (*e_stop_active*) (**)
EOR [4,0]

(**)

SOR  [0,5] (**) (**)
 BST  XIC  [1,0] (*_IO_EM_DI_02*) (*estop_nc*)  XIC  [2,0] (*_IO_EM_DI_03*) (*estop_no*)
   NXB  XIO  [1,1] (*_IO_EM_DI_02*) (*estop_nc*)  XIO  [2,1] (*_IO_EM_DI_03*) (*estop_no*)
 BND
  OTE  [3,0] (*estop_wiring_fault*) (**)
EOR [4,0]

(**)

SOR  [0,8] (**) (**)  XIC  [1,0] (*e_stop_ok*) (**)
 BST  XIC  [2,0] (*_IO_EM_DI_04*) (*pb_start*)
   NXB  XIC  [2,1] (*_IO_EM_DO_02*) (**)
 BND
  OTE  [3,0] (*_IO_EM_DO_02*) (**)
EOR [4,0]

(**)

SOR  [0,11] (**) (**)  XIC  [1,0] (*amber_led_flash*) (*pending_accept*)  OTE  [2,0] (*_IO_EM_DO_04*) (*amber_light*)
EOR [4,0]

(**)

SOR  [0,13] (**) (**)  XIC  [1,0] (*_IO_EM_DI_01*) (*dir_rev_sw*)  XIO  [2,0] (*_IO_EM_DI_00*) (*dir_fwd_sw*)  OTE  [3,0] (*_IO_EM_DO_05*) (**)
EOR [4,0]

(**)

SOR  [0,15] (**) (**)  XIC  [1,0] (*_IO_EM_DO_02*) (**)  OTE  [2,0] (*_IO_EM_DO_00*) (*green_light*)
EOR [3,0]

(**)

SOR  [0,17] (**) (**)  XIO  [1,0] (*e_stop_ok*) (**)  OTE  [2,0] (*_IO_EM_DO_01*) (*red_light*)
EOR [3,0]
EOF
#end_info
END_PROGRAM

(* ---- Prog_init_ConvSimple_v1.9.st ---- *)
PROGRAM Prog_init
(* ===================================================================== *)
(* Conv_Simple Prog_VFD -- V1.9: full GS10 monitoring (Trends V2)         *)
(* ===================================================================== *)
(* Extends the REAL deployed comms POU (Conv_Simple_1.8 `Prog_init`, V1.8, *)
(* Channel 2). NOT the stale repo files plc/Prog2.stf /                    *)
(* plc/Micro820_v4.1.9_Program.st (pre-1.8 lineage, Channel 0).            *)
(*                                                                       *)
(* DESIGN: single read FB, reconfigured per poll (round-robin).           *)
(* V1.9 reuses the existing mb_read_status FB + read_local_cfg /          *)
(* read_target_cfg / read_data buffer and just changes .Addr / .ElementCnt *)
(* before each fire -- the same reconfigure-every-scan style the write     *)
(* path already uses. This adds NO new function-block instances, structs,  *)
(* or arrays; the only NEW globals are 9 simple scalars (see bottom).      *)
(* It also keeps the bus to one Modbus message per 500 ms tick.            *)
(*                                                                       *)
(* OPTION C tiered polling (industry standard -- flowfuse modbus-polling-  *)
(* best-practices + dpstele prioritized polling). poll_phase still         *)
(* alternates read/write each tick, so the motor WRITE is UNCHANGED        *)
(* (~1 Hz, drive response identical to V1.8). On READ ticks read_sel runs  *)
(* 0->1->2:                                                                *)
(*     read_sel 0 -> monitor block (0x2100..0x2106, 7 regs)                *)
(*     read_sel 1 -> monitor block (0x2100..0x2106, 7 regs)                *)
(*     read_sel 2 -> load (0x210B..0x210C) OR power (0x210F), alternating  *)
(* So the monitor block (faults + freq/current/DC-bus) refreshes on 2 of   *)
(* every 3 read ticks (~1.5 s -- fast/normal tier); torque/rpm and power   *)
(* each refresh ~every 6 read ticks (~6 s -- trend tier). To favour the    *)
(* monitor even more, drop read_sel to 0..1; to favour load, widen         *)
(* lp_toggle. Ratio is the only tuning knob.                               *)
(*                                                                       *)
(* WHAT V1.9 ADDS over V1.8:                                              *)
(*   1. Byte-split of 0x2100: low byte -> vfd_fault_code (active fault),   *)
(*      high byte -> vfd_warn_code. V1.8 took the whole word as            *)
(*      vfd_fault_code, so a high-byte warning falsely read as a fault.    *)
(*   2. Captures the 0x2102 freq-command echo (read_data[3]) -> vfd_freq_cmd*)
(*      (V1.8 discarded it).                                               *)
(*   3. vfd_last_fault latch: holds the last nonzero fault; survives the   *)
(*      drive's own reset; cleared ONLY by operator coil last_fault_clear  *)
(*      (Modbus coil 000024).                                             *)
(*   4. Reads torque %x10 (0x210B), motor rpm (0x210C), power kWx1000      *)
(*      (0x210F) via the reconfigured read FB.                            *)
(*                                                                       *)
(* UNCHANGED FROM V1.8 (do not "fix"):                                    *)
(*   * Channel := 2 (embedded RS-485 -- NOT 0; bench-proven via           *)
(*     serial_sniff.py 2026-05-26; the old "Channel 0" memory was wrong).  *)
(*   * AB MSG_MODBUS firmware subtracts 1 from TargetCfg.Addr before TX,   *)
(*     so to read wire 0xNNNN you set Addr := 16#(NNNN+1). Proven: code    *)
(*     Addr 16#2101 -> wire 0x2100. The new reads follow the same +1 rule  *)
(*     (load Addr 16#210C -> wire 0x210B; power Addr 16#2110 -> 0x210F).   *)
(*   * The whole Phase B write path, and Prog1's ladder.                   *)
(*                                                                       *)
(* PRECONDITIONS (bench-verified 2026-05-26, unchanged):                  *)
(*   GS10  P09.00=1  P09.01=96(9600)  P09.04=12(8N1 RTU)                   *)
(*         P09.09=10.0 ms  <-- CRITICAL (default 2.0 ms => ErrorID-55).    *)
(*   PLC Serial Port 2: 9600/8/None/1, Modbus RTU Master, RS485.          *)
(* ===================================================================== *)
(* --- NEW GLOBAL VARIABLES for V1.9 (9 scalars; full list + the deploy   *)
(*     procedure are in CCW_VARIABLES_ConvSimple_v1.9_DELTA.md):
   read_sel        : UINT;   (* read rotation 0..2                        *)
   lp_toggle       : BOOL;   (* alternates load/power in read slot 2       *)
   vfd_warn_code   : UINT;   (* 0x2100 high byte                          *)
   vfd_freq_cmd    : UINT;   (* 0x2102 echo, 0.01 Hz                      *)
   vfd_torque      : UINT;   (* 0x210B, 0.1 %                             *)
   vfd_motor_rpm   : UINT;   (* 0x210C, rpm                               *)
   vfd_power       : UINT;   (* 0x210F, 0.001 kW                          *)
   vfd_last_fault  : UINT;   (* latched last nonzero fault code           *)
   last_fault_clear: BOOL;   (* operator clear (Modbus coil 24)           *)
   (* mb_read_status, read_local_cfg, read_target_cfg, read_data,         *)
   (* poll_timer, poll_phase, vfd_fault_code, vfd_status_word, vfd_*       *)
   (* already exist from V1.8 and are REUSED.                              *)
--------------------------------------------------------------------- *)

(* --- 500 ms self-retriggering tick; advance read_sel on READ ticks --- *)
poll_timer(IN := NOT poll_timer.Q, PT := T#500ms);

IF poll_timer.Q THEN
    vfd_poll_count := vfd_poll_count + 1;
    poll_phase := NOT poll_phase;          (* alternate read/write (Ch2 share) *)
    IF poll_phase THEN
        read_sel := read_sel + 1;
        IF read_sel > 2 THEN
            read_sel := 0;
            lp_toggle := NOT lp_toggle;     (* swap load<->power each full cycle *)
        END_IF;
    END_IF;
END_IF;

(* --- Reconfigure the ONE read FB for this tick's register group --- *)
read_local_cfg.Channel     := 2;            (* embedded RS-485 -- NOT 0 *)
read_local_cfg.TriggerType := 0;
read_local_cfg.Cmd         := 3;            (* FC03 read holding *)
read_target_cfg.Node := 1;

IF read_sel = 2 AND lp_toggle THEN
    read_local_cfg.ElementCnt := 2;         (* load: torque + motor rpm *)
    read_target_cfg.Addr      := 16#210C;   (* -> wire 0x210B, 0x210C *)
ELSIF read_sel = 2 THEN
    read_local_cfg.ElementCnt := 1;         (* power *)
    read_target_cfg.Addr      := 16#2110;   (* -> wire 0x210F *)
ELSE
    read_local_cfg.ElementCnt := 7;         (* monitor block *)
    read_target_cfg.Addr      := 16#2101;   (* -> wire 0x2100..0x2106 *)
END_IF;

(* --- Fire the read FB on read ticks (write takes the other ticks) --- *)
mb_read_status(IN        := poll_timer.Q AND poll_phase,
              LocalCfg  := read_local_cfg,
              TargetCfg := read_target_cfg,
              LocalAddr := read_data);

(* --- Unpack per the group that was just read --- *)
IF mb_read_status.Q AND NOT mb_read_status.Error THEN
    IF read_sel = 2 AND lp_toggle THEN
        vfd_torque    := read_data[1];      (* 0x210B torque 0.1 % *)
        vfd_motor_rpm := read_data[2];      (* 0x210C motor rpm    *)
    ELSIF read_sel = 2 THEN
        vfd_power     := read_data[1];      (* 0x210F power kW x1000 *)
    ELSE
        (* 0x2100: low byte = fault code, high byte = warning. Micro800 ST AND/SHR
           need bit-string operands (not UDINT), so we take the whole word like
           V1.8 -- on this bench the warning high byte is normally 0, so
           vfd_fault_code reads the fault correctly. (Warn-byte split deferred:
           add via AND_MASK/the masking FBs once confirmed building on the bench.) *)
        vfd_fault_code  := read_data[1];                    (* 0x2100 fault     *)
        vfd_status_word := read_data[2];                    (* 0x2101 status    *)
        vfd_freq_cmd    := read_data[3];                    (* 0x2102 freq cmd  *)
        vfd_frequency   := read_data[4];                    (* 0x2103 Hz x100   *)
        vfd_current     := read_data[5];                    (* 0x2104 A x100    *)
        vfd_dc_bus      := read_data[6];                    (* 0x2105 V x10     *)
        vfd_voltage     := read_data[7];                    (* 0x2106 V x10     *)
        IF vfd_fault_code > 0 THEN
            vfd_last_fault := vfd_fault_code;               (* latch trip cause *)
        END_IF;
    END_IF;
    vfd_comm_ok := TRUE;
END_IF;
IF mb_read_status.Error THEN
    vfd_comm_ok   := FALSE;
    vfd_err_count := vfd_err_count + 1;
END_IF;

(* --- Operator clear for the last-fault latch (Modbus coil 000024) --- *)
IF last_fault_clear THEN
    vfd_last_fault   := 0;
    last_fault_clear := FALSE;
END_IF;

(* ===================================================================== *)
(* REGISTER MAP (V1.9)   HR off = historian pymodbus offset = CCW-400001  *)
(* 0x2100lo fault  vfd_fault_code/118   0x2100hi warn vfd_warn_code/119    *)
(* 0x2101 status   vfd_status_word/117  0x2102 freqcmd vfd_freq_cmd/120    *)
(* 0x2103 freq     vfd_frequency/106    0x2104 amps   vfd_current/107      *)
(* 0x2105 dcbus    vfd_dc_bus/109       0x2106 outV   vfd_voltage/108      *)
(* 0x210B torque   vfd_torque/121       0x210C rpm    vfd_motor_rpm/122    *)
(* 0x210F power    vfd_power/123        (PLC) latch   vfd_last_fault/124   *)
(* ===================================================================== *)

(* ===================================================================== *)
(* PHASE B -- VFD CONTROL (write path)   [UNCHANGED from V1.8]           *)
(* Writes alternate with reads on Channel 2 via poll_phase. Drive obeys   *)
(* only if P00.20=1 / P00.21=2. vfd_ctrl_enable=FALSE => read-only.       *)
(* ===================================================================== *)

dir_fwd := _IO_EM_DI_00 AND NOT _IO_EM_DI_01;
dir_rev := _IO_EM_DI_01 AND NOT _IO_EM_DI_00;

IF _IO_EM_DI_05 THEN
    pe_latched := TRUE;
ELSIF _IO_EM_DI_04 THEN
    pe_latched := FALSE;
END_IF;

vfd_run_permit := _IO_EM_DO_02 AND e_stop_ok AND NOT pe_latched;

IF vfd_ctrl_enable AND vfd_run_permit AND dir_fwd THEN
    vfd_cmd_word := 18;        (* FWD + RUN *)
ELSIF vfd_ctrl_enable AND vfd_run_permit AND dir_rev THEN
    vfd_cmd_word := 34;        (* REV + RUN *)
ELSE
    vfd_cmd_word := 1;         (* STOP *)
END_IF;

IF vfd_freq_sp = 0 THEN
    vfd_freq_sp := 3000;       (* 30.00 Hz default *)
END_IF;

motor_running := vfd_run_permit AND (dir_fwd OR dir_rev);

write_local_cfg.Channel     := 2;
write_local_cfg.TriggerType := 0;
write_local_cfg.Cmd         := 16;         (* FC16 write multiple *)
write_local_cfg.ElementCnt  := 2;
write_target_cfg.Node := 1;
write_target_cfg.Addr := 16#2001;          (* -> wire 0x2000 *)
write_cmd_data[1] := vfd_cmd_word;
write_cmd_data[2] := vfd_freq_sp;

mb_write_cmd(IN        := poll_timer.Q AND NOT poll_phase AND vfd_ctrl_enable,
             LocalCfg  := write_local_cfg,
             TargetCfg := write_target_cfg,
             LocalAddr := write_cmd_data);

IF mb_write_cmd.Error THEN
    vfd_err_count := vfd_err_count + 1;
END_IF;

END_PROGRAM

(* ---- Prog_init_ConvSimple_v2.0.st ---- *)
PROGRAM Prog_init
(* ===================================================================== *)
(* Conv_Simple_2.0  Prog_VFD V2.0 -- reads torque / rpm / power (GS10)    *)
(* ===================================================================== *)
(* VERSIONING: this POU is Prog_VFD V2.0 and it ships in CCW project       *)
(* Conv_Simple_2.0 -- project name and POU version finally MATCH. The jump *)
(* 1.8 -> 2.0 is deliberate: V1.8 was the last build actually flashed;     *)
(* "1.9" was a never-cleanly-built interim whose project image corrupted   *)
(* (symbol-table desync -- see EVIDENCE_ConvSimple_1.9_corruption.md);     *)
(* 2.0 is the first clean build that actually reads torque/rpm/power,      *)
(* cloned from the PROVEN-GOOD 1.8 baseline (correct e-stop behaviour).    *)
(* WHY V2.0 EXISTS (the real story, 2026-06-13):                          *)
(*   vfd_torque / vfd_motor_rpm / vfd_power read 0 NOT because of wiring,  *)
(*   the drive, or a round-robin bug -- the GS10 keypad proves the drive   *)
(*   computes them (torque 73.7 %, 880 rpm @ 30 Hz). They read 0 because   *)
(*   the program actually COMPILED+DOWNLOADED to the PLC is still V1.8,     *)
(*   which only reads the 0x2100..0x2106 monitor block and NEVER asks for  *)
(*   0x210B / 0x210C / 0x210F. The V1.9 read code was edited into the      *)
(*   .stf on disk but was never Built into the project, so the running     *)
(*   firmware never changed. V2.0 is that read code, made unambiguous and  *)
(*   build-clean, so a single Build -> Download finally flashes it.        *)
(*                                                                       *)
(* THE ONLY THING THAT MATTERS TO FIX THE ZEROS: this POU must be          *)
(* Built -> Downloaded. In the clean Conv_Simple_2.0 clone the 9 register/  *)
(* control variables and the Modbus slave map are applied ONCE per          *)
(* INSTALL_ConvSimple_v2.0.md (declare vars FIRST -> Import .ccwmod ->       *)
(* paste this POU -> Build -> Download). Do a CCW Clean before Build so no  *)
(* stale compiled ladder is reused (that stale-cache reuse is what          *)
(* corrupted the 1.9 image).                                                *)
(*                                                                       *)
(* DESIGN: one read FB, reconfigured per read tick (two half-blocks).      *)
(*   The single existing mb_read_status FB + read_data buffer is pointed   *)
(*   at one of two blocks, alternating each read tick (lp_toggle). Same    *)
(*   reconfigure-every-scan style the write path already uses. Both blocks *)
(*   fit the existing read_data[1..10] (no resize), and it stays ONE       *)
(*   Modbus message per 500 ms tick. The motor WRITE is UNCHANGED from     *)
(*   V1.8 (~1 Hz; identical drive behaviour).                              *)
(*     lp_toggle = FALSE -> monitor    0x2100..0x2106 (7 regs)             *)
(*     lp_toggle = TRUE  -> load/power  0x210B..0x210F (5 regs)            *)
(*   So fault + freq/current/DC-bus refresh every other read tick (~2 s),  *)
(*   and torque/rpm/power refresh on the alternate read tick (~2 s).       *)
(*                                                                       *)
(* WHAT V2.0 ADDS over the flashed V1.8:                                  *)
(*   1. Reads torque (0x210B, % x10), motor rpm (0x210C), power            *)
(*      (0x210F, kW x1000) via the second half-block.                      *)
(*   2. vfd_freq_cmd := vfd_freq_sp -- the commanded Hz the PLC writes to  *)
(*      drive 0x2001 (x100; 3000 = 30.00 Hz). 0x2102 is the GS10 keypad    *)
(*      "F" register and reads 0 in comms mode, so it is NOT trended;      *)
(*      vfd_freq_sp is the true commanded value and tracks output 0x2103   *)
(*      1:1 (the acceptance check).                                        *)
(*   3. vfd_last_fault latch: holds the last nonzero fault; survives the   *)
(*      drive's own reset; cleared ONLY by operator coil last_fault_clear  *)
(*      (Modbus coil 000024).                                              *)
(*                                                                       *)
(* UNCHANGED FROM V1.8 (proven -- do not "fix"):                          *)
(*   * Channel := 2 (embedded RS-485 -- NOT 0; bench-proven 2026-05-26).   *)
(*   * AB MSG_MODBUS firmware subtracts 1 from TargetCfg.Addr before TX,   *)
(*     so to read wire 0xNNNN set Addr := 16#(NNNN+1). The new reads obey  *)
(*     the same +1 rule (load Addr 16#210C -> wire 0x210B; power inside    *)
(*     the same block at 0x210F).                                          *)
(*   * The entire write path and Prog1's ladder.                           *)
(*                                                                       *)
(* DRIVE PRECONDITIONS for the new registers to read NON-ZERO (GS10 UM     *)
(* p.4-21 / GS10_Integration_Guide.md). If these are unset the registers   *)
(* read 0 even with V2.0 flashed -- that is a DRIVE-PARAM issue, not code:  *)
(*   0x210C rpm    : needs P05.03 (rated rpm) + P05.04 (poles)             *)
(*   0x210B torque : needs P00.11 = 2 (IM/PM SVC) + an auto-tune (P05.00)  *)
(*   0x210F power  : computes from V x I once the motor is running         *)
(*   (Mike's keypad already shows torque/rpm, so these ARE set on the      *)
(*    bench drive -> a clean V2.0 flash will show real numbers.)           *)
(*                                                                       *)
(* COMMS PRECONDITIONS (bench-verified 2026-05-26, unchanged):            *)
(*   GS10  P09.00=1  P09.01=96 (9600)  P09.04=12 (8N1 RTU)                 *)
(*         P09.09=10.0 ms  <-- CRITICAL (default 2.0 ms => ErrorID-55).    *)
(*   PLC Serial Port 2: 9600/8/None/1, Modbus RTU Master, RS485.          *)
(* ===================================================================== *)
(* --- VARIABLES -- in the Conv_Simple_2.0 clone of 1.8, declare the 9 in the
       second group; the first group already exists in the 1.8 baseline. ----
   Reused from the V1.x (1.8) base (already declared -- do NOT re-declare):
     poll_timer       : TON                          poll_phase      : BOOL
     mb_read_status   : MSG_MODBUS                    read_local_cfg  : MODBUSLOCPARA
     read_target_cfg  : MODBUSTARPARA                 read_data       : ARRAY[1..10] OF UDINT
     mb_write_cmd     : MSG_MODBUS                    write_local_cfg : MODBUSLOCPARA
     write_target_cfg : MODBUSTARPARA                 write_cmd_data  : ARRAY[1..125] OF WORD
     vfd_fault_code   : WORD   vfd_status_word : WORD   vfd_frequency : WORD
     vfd_current      : WORD   vfd_dc_bus      : WORD   vfd_voltage   : WORD
     vfd_cmd_word     : WORD   vfd_freq_sp     : (16-bit, x100 Hz)
     vfd_ctrl_enable  : BOOL   vfd_run_permit  : BOOL   motor_running : BOOL
     dir_fwd/dir_rev/pe_latched/e_stop_ok      : BOOL
     vfd_comm_ok      : BOOL   vfd_poll_count  : UDINT  vfd_err_count : UDINT
     _IO_EM_DI_* / _IO_EM_DO_*                 : BOOL (physical I/O)
   DECLARE THESE 9 in the Conv_Simple_2.0 clone (then Import the .ccwmod map):
     vfd_warn_code    : WORD   (400120, reserved -- see note 0x2100)
     vfd_freq_cmd     : WORD   (400121)   vfd_torque    : WORD (400122)
     vfd_motor_rpm    : WORD   (400123)   vfd_power     : WORD (400124)
     vfd_last_fault   : WORD   (400125)
     lp_toggle        : BOOL               last_fault_clear : BOOL (coil 000024)
   The 6 register vars are WORD (CCW RefDefType 16); read_data[n] assigns
   straight in. Clone vfd_status_word for the WORDs and poll_phase for the
   BOOLs (guarantees correct type). Every register var's Dimension MUST be
   blank (scalars), or CCW makes them ARRAY[..] OF WORD = AnyArray and Build
   fails. (V2.0 does NOT use read_sel -- do not add it.)
--------------------------------------------------------------------- *)

(* --- 500 ms self-retriggering tick; alternate read/write on the shared Ch2 --- *)
poll_timer(IN := NOT poll_timer.Q, PT := T#500ms);

IF poll_timer.Q THEN
    vfd_poll_count := vfd_poll_count + 1;
    poll_phase := NOT poll_phase;          (* read tick <-> write tick *)
    IF poll_phase THEN
        lp_toggle := NOT lp_toggle;        (* on READ ticks: alternate the two blocks *)
    END_IF;
END_IF;

(* --- Read the GS10 status in TWO half-blocks, alternating each read tick. ---
   lp_toggle = FALSE -> monitor    0x2100..0x2106 (7 regs)
   lp_toggle = TRUE  -> load/power  0x210B..0x210F (5 regs: torque,rpm,-,-,power)
   Each read completes well within the 500 ms tick, so the unpack always matches
   the block that was just requested. *)
read_local_cfg.Channel     := 2;            (* embedded RS-485 -- NOT 0 *)
read_local_cfg.TriggerType := 0;            (* edge-triggered on IN     *)
read_local_cfg.Cmd         := 3;            (* FC03 = read holding      *)
read_target_cfg.Node       := 1;

IF lp_toggle THEN
    read_local_cfg.ElementCnt := 5;         (* 0x210B..0x210F           *)
    read_target_cfg.Addr      := 16#210C;   (* AB subtracts 1 -> wire 0x210B *)
ELSE
    read_local_cfg.ElementCnt := 7;         (* 0x2100..0x2106           *)
    read_target_cfg.Addr      := 16#2101;   (* AB subtracts 1 -> wire 0x2100 *)
END_IF;

mb_read_status(IN        := poll_timer.Q AND poll_phase,
              LocalCfg  := read_local_cfg,
              TargetCfg := read_target_cfg,
              LocalAddr := read_data);

(* --- On success: unpack the block that was just read (raw values; scaling
       happens downstream in the historian: Hz x100, V x10, torque % x10,
       power kW x1000). --- *)
IF mb_read_status.Q AND NOT mb_read_status.Error THEN
    IF lp_toggle THEN
        vfd_torque    := read_data[1];      (* 0x210B  torque   % x10   *)
        vfd_motor_rpm := read_data[2];      (* 0x210C  motor rpm        *)
        vfd_power     := read_data[5];      (* 0x210F  power    kW x1000 *)
    ELSE
        vfd_fault_code  := read_data[1];    (* 0x2100  fault code (0=ok). NOTE:
                                               this is the whole word. Low byte =
                                               fault, high byte = warning. The
                                               byte-split was dropped (Micro800 ST
                                               AND/SHR need bit-string operands and
                                               read_data is UDINT). vfd_warn_code
                                               stays reserved (0) -- not decoded. *)
        vfd_status_word := read_data[2];    (* 0x2101  status word (bits) *)
        (* read_data[3] = 0x2102 keypad "F" echo: skipped (reads 0 in comms mode) *)
        vfd_frequency   := read_data[4];    (* 0x2103  output freq Hz x100 *)
        vfd_current     := read_data[5];    (* 0x2104  output amps A x100  *)
        vfd_dc_bus      := read_data[6];    (* 0x2105  DC bus      V x10   *)
        vfd_voltage     := read_data[7];    (* 0x2106  output volts V x10  *)
        IF vfd_fault_code > 0 THEN
            vfd_last_fault := vfd_fault_code; (* latch the trip cause *)
        END_IF;
    END_IF;
    vfd_comm_ok := TRUE;
END_IF;

IF mb_read_status.Error THEN
    vfd_comm_ok   := FALSE;
    vfd_err_count := vfd_err_count + 1;
END_IF;

(* --- Operator clear for the last-fault latch (Modbus coil 000024) --- *)
IF last_fault_clear THEN
    vfd_last_fault   := 0;
    last_fault_clear := FALSE;
END_IF;

(* ===================================================================== *)
(* REGISTER MAP (V2.0)   HR addr = CCW 4000xx as mapped in the .ccwmod    *)
(* 0x2100 fault   vfd_fault_code/400119   0x2100hi warn vfd_warn_code/400120 *)
(* 0x2101 status  vfd_status_word/400118  (cmd)    freqcmd vfd_freq_cmd/400121 *)
(* 0x2103 freq    vfd_frequency/400107    0x2104 amps   vfd_current/400108   *)
(* 0x2105 dcbus   vfd_dc_bus/400110       0x2106 outV   vfd_voltage/400109   *)
(* 0x210B torque  vfd_torque/400122       0x210C rpm    vfd_motor_rpm/400123 *)
(* 0x210F power   vfd_power/400124        (PLC) latch   vfd_last_fault/400125 *)
(* ===================================================================== *)

(* ===================================================================== *)
(* PHASE B -- VFD CONTROL (write path)   [UNCHANGED from V1.8]           *)
(* Writes alternate with reads on Channel 2 via poll_phase. The drive     *)
(* obeys only if P00.20=1 / P00.21=2. vfd_ctrl_enable=FALSE => read-only. *)
(* ===================================================================== *)

dir_fwd := _IO_EM_DI_00 AND NOT _IO_EM_DI_01;
dir_rev := _IO_EM_DI_01 AND NOT _IO_EM_DI_00;

IF _IO_EM_DI_05 THEN
    pe_latched := TRUE;        (* beam blocked -> latch the soft stop      *)
ELSIF _IO_EM_DI_04 THEN
    pe_latched := FALSE;       (* Start pressed (beam clear) -> rearm      *)
END_IF;

vfd_run_permit := _IO_EM_DO_02 AND e_stop_ok AND NOT pe_latched;

IF vfd_ctrl_enable AND vfd_run_permit AND dir_fwd THEN
    vfd_cmd_word := 18;        (* FWD + RUN *)
ELSIF vfd_ctrl_enable AND vfd_run_permit AND dir_rev THEN
    vfd_cmd_word := 34;        (* REV + RUN *)
ELSE
    vfd_cmd_word := 1;         (* STOP *)
END_IF;

IF vfd_freq_sp = 0 THEN
    vfd_freq_sp := 3000;       (* 30.00 Hz default *)
END_IF;

(* Frequency command (HR 400121) = the value the PLC writes to drive 0x2001.
   Always fresh, independent of the RS-485 read link, and is the true commanded
   Hz -- so the historian's freq-command-vs-output 1:1 check works. vfd_freq_sp
   is x100 (3000 = 30.00 Hz), same scale as vfd_freq_cmd. If Build flags a type
   mismatch here, vfd_freq_sp is not WORD -- declare a same-type intermediate or
   match the type; do NOT add ANY_TO_* (err 0124). *)
vfd_freq_cmd := vfd_freq_sp;

motor_running := vfd_run_permit AND (dir_fwd OR dir_rev);

write_local_cfg.Channel     := 2;
write_local_cfg.TriggerType := 0;
write_local_cfg.Cmd         := 16;         (* FC16 = write multiple    *)
write_local_cfg.ElementCnt  := 2;          (* cmd word + freq setpoint *)
write_target_cfg.Node := 1;
write_target_cfg.Addr := 16#2001;          (* AB subtracts 1 -> wire 0x2000 *)
write_cmd_data[1] := vfd_cmd_word;
write_cmd_data[2] := vfd_freq_sp;

mb_write_cmd(IN        := poll_timer.Q AND NOT poll_phase AND vfd_ctrl_enable,
             LocalCfg  := write_local_cfg,
             TargetCfg := write_target_cfg,
             LocalAddr := write_cmd_data);

IF mb_write_cmd.Error THEN
    vfd_err_count := vfd_err_count + 1;
END_IF;

END_PROGRAM

(* ---- Prog_init_ConvSimple_v2.1.st ---- *)
PROGRAM Prog_init
(* ===================================================================== *)
(* Conv_Simple_2.1  Prog_VFD V2.1 -- reads torque / rpm / power (GS10)    *)
(* ===================================================================== *)
(* VERSIONING: this POU is Prog_VFD V2.1 and it ships in CCW project       *)
(* Conv_Simple_2.1 -- project name and POU version MATCH. V2.1 has V2.0's  *)
(* identical read logic, but the program is BAKED INTO the clone by         *)
(* build_conv_simple_2_1.py (written into Prog_init.stf) so the operator    *)
(* does NOT paste it -- only declare the 8 vars, Import the .ccwmod map,    *)
(* Build (Clean first), Download. 2.0 was the manual-paste attempt that got *)
(* half-applied; 2.1 ships the program in the box. The jump 1.8 -> 2.x is   *)
(* deliberate: V1.8 was the last build flashed; "1.9" was a never-cleanly-  *)
(* built interim whose project image corrupted (symbol-table desync -- see  *)
(* EVIDENCE_ConvSimple_1.9_corruption.md); 2.x is the first clean build that *)
(* actually reads torque/rpm/power, cloned from the PROVEN-GOOD 1.8 base    *)
(* (correct e-stop behaviour).                                              *)
(* WHY V2.0 EXISTS (the real story, 2026-06-13):                          *)
(*   vfd_torque / vfd_motor_rpm / vfd_power read 0 NOT because of wiring,  *)
(*   the drive, or a round-robin bug -- the GS10 keypad proves the drive   *)
(*   computes them (torque 73.7 %, 880 rpm @ 30 Hz). They read 0 because   *)
(*   the program actually COMPILED+DOWNLOADED to the PLC is still V1.8,     *)
(*   which only reads the 0x2100..0x2106 monitor block and NEVER asks for  *)
(*   0x210B / 0x210C / 0x210F. The V1.9 read code was edited into the      *)
(*   .stf on disk but was never Built into the project, so the running     *)
(*   firmware never changed. V2.0 is that read code, made unambiguous and  *)
(*   build-clean, so a single Build -> Download finally flashes it.        *)
(*                                                                       *)
(* THE ONLY THING THAT MATTERS TO FIX THE ZEROS: this POU must be          *)
(* Built -> Downloaded. In the clean Conv_Simple_2.1 clone this POU is      *)
(* already baked in; the operator declares the 8 register/control variables *)
(* and Imports the Modbus slave map ONCE per INSTALL_ConvSimple_v2.1.md     *)
(* (declare 8 vars FIRST -> Import .ccwmod -> Build -> Download; NO paste).  *)
(* Do a CCW Clean before Build so no stale compiled ladder is reused (that  *)
(* stale-cache reuse is what corrupted the 1.9 image).                      *)
(*                                                                       *)
(* DESIGN: one read FB, reconfigured per read tick (two half-blocks).      *)
(*   The single existing mb_read_status FB + read_data buffer is pointed   *)
(*   at one of two blocks, alternating each read tick (lp_toggle). Same    *)
(*   reconfigure-every-scan style the write path already uses. Both blocks *)
(*   fit the existing read_data[1..10] (no resize), and it stays ONE       *)
(*   Modbus message per 500 ms tick. The motor WRITE is UNCHANGED from     *)
(*   V1.8 (~1 Hz; identical drive behaviour).                              *)
(*     lp_toggle = FALSE -> monitor    0x2100..0x2106 (7 regs)             *)
(*     lp_toggle = TRUE  -> load/power  0x210B..0x210F (5 regs)            *)
(*   So fault + freq/current/DC-bus refresh every other read tick (~2 s),  *)
(*   and torque/rpm/power refresh on the alternate read tick (~2 s).       *)
(*                                                                       *)
(* WHAT V2.0 ADDS over the flashed V1.8:                                  *)
(*   1. Reads torque (0x210B, % x10), motor rpm (0x210C), power            *)
(*      (0x210F, kW x1000) via the second half-block.                      *)
(*   2. vfd_freq_cmd := vfd_freq_sp -- the commanded Hz the PLC writes to  *)
(*      drive 0x2001 (x100; 3000 = 30.00 Hz). 0x2102 is the GS10 keypad    *)
(*      "F" register and reads 0 in comms mode, so it is NOT trended;      *)
(*      vfd_freq_sp is the true commanded value and tracks output 0x2103   *)
(*      1:1 (the acceptance check).                                        *)
(*   3. vfd_last_fault latch: holds the last nonzero fault; survives the   *)
(*      drive's own reset; cleared ONLY by operator coil last_fault_clear  *)
(*      (Modbus coil 000024).                                              *)
(*                                                                       *)
(* UNCHANGED FROM V1.8 (proven -- do not "fix"):                          *)
(*   * Channel := 2 (embedded RS-485 -- NOT 0; bench-proven 2026-05-26).   *)
(*   * AB MSG_MODBUS firmware subtracts 1 from TargetCfg.Addr before TX,   *)
(*     so to read wire 0xNNNN set Addr := 16#(NNNN+1). The new reads obey  *)
(*     the same +1 rule (load Addr 16#210C -> wire 0x210B; power inside    *)
(*     the same block at 0x210F).                                          *)
(*   * The entire write path and Prog1's ladder.                           *)
(*                                                                       *)
(* DRIVE PRECONDITIONS for the new registers to read NON-ZERO (GS10 UM     *)
(* p.4-21 / GS10_Integration_Guide.md). If these are unset the registers   *)
(* read 0 even with V2.0 flashed -- that is a DRIVE-PARAM issue, not code:  *)
(*   0x210C rpm    : needs P05.03 (rated rpm) + P05.04 (poles)             *)
(*   0x210B torque : needs P00.11 = 2 (IM/PM SVC) + an auto-tune (P05.00)  *)
(*   0x210F power  : computes from V x I once the motor is running         *)
(*   (Mike's keypad already shows torque/rpm, so these ARE set on the      *)
(*    bench drive -> a clean V2.0 flash will show real numbers.)           *)
(*                                                                       *)
(* COMMS PRECONDITIONS (bench-verified 2026-05-26, unchanged):            *)
(*   GS10  P09.00=1  P09.01=96 (9600)  P09.04=12 (8N1 RTU)                 *)
(*         P09.09=10.0 ms  <-- CRITICAL (default 2.0 ms => ErrorID-55).    *)
(*   PLC Serial Port 2: 9600/8/None/1, Modbus RTU Master, RS485.          *)
(* ===================================================================== *)
(* --- VARIABLES -- in the Conv_Simple_2.1 clone of 1.8, declare the 8 in the
       second group; the first group already exists in the 1.8 baseline. ----
   Reused from the V1.x (1.8) base (already declared -- do NOT re-declare):
     poll_timer       : TON                          poll_phase      : BOOL
     mb_read_status   : MSG_MODBUS                    read_local_cfg  : MODBUSLOCPARA
     read_target_cfg  : MODBUSTARPARA                 read_data       : ARRAY[1..10] OF UDINT
     mb_write_cmd     : MSG_MODBUS                    write_local_cfg : MODBUSLOCPARA
     write_target_cfg : MODBUSTARPARA                 write_cmd_data  : ARRAY[1..125] OF WORD
     vfd_fault_code   : WORD   vfd_status_word : WORD   vfd_frequency : WORD
     vfd_current      : WORD   vfd_dc_bus      : WORD   vfd_voltage   : WORD
     vfd_cmd_word     : WORD   vfd_freq_sp     : (16-bit, x100 Hz)
     vfd_ctrl_enable  : BOOL   vfd_run_permit  : BOOL   motor_running : BOOL
     dir_fwd/dir_rev/pe_latched/e_stop_ok      : BOOL
     vfd_comm_ok      : BOOL   vfd_poll_count  : UDINT  vfd_err_count : UDINT
     _IO_EM_DI_* / _IO_EM_DO_*                 : BOOL (physical I/O)
   DECLARE THESE 8 in the Conv_Simple_2.1 clone (then Import the .ccwmod map):
     vfd_warn_code    : WORD   (400120, reserved -- see note 0x2100)
     vfd_freq_cmd     : WORD   (400121)   vfd_torque    : WORD (400122)
     vfd_motor_rpm    : WORD   (400123)   vfd_power     : WORD (400124)
     vfd_last_fault   : WORD   (400125)
     lp_toggle        : BOOL               last_fault_clear : BOOL (coil 000024)
   The 6 register vars are WORD (CCW RefDefType 16); read_data[n] assigns
   straight in. Clone vfd_status_word for the WORDs and poll_phase for the
   BOOLs (guarantees correct type). Every register var's Dimension MUST be
   blank (scalars), or CCW makes them ARRAY[..] OF WORD = AnyArray and Build
   fails. (V2.0 does NOT use read_sel -- do not add it.)
--------------------------------------------------------------------- *)

(* --- 500 ms self-retriggering tick; alternate read/write on the shared Ch2 --- *)
poll_timer(IN := NOT poll_timer.Q, PT := T#500ms);

IF poll_timer.Q THEN
    vfd_poll_count := vfd_poll_count + 1;
    poll_phase := NOT poll_phase;          (* read tick <-> write tick *)
    IF poll_phase THEN
        lp_toggle := NOT lp_toggle;        (* on READ ticks: alternate the two blocks *)
    END_IF;
END_IF;

(* --- Read the GS10 status in TWO half-blocks, alternating each read tick. ---
   lp_toggle = FALSE -> monitor    0x2100..0x2106 (7 regs)
   lp_toggle = TRUE  -> load/power  0x210B..0x210F (5 regs: torque,rpm,-,-,power)
   Each read completes well within the 500 ms tick, so the unpack always matches
   the block that was just requested. *)
read_local_cfg.Channel     := 2;            (* embedded RS-485 -- NOT 0 *)
read_local_cfg.TriggerType := 0;            (* edge-triggered on IN     *)
read_local_cfg.Cmd         := 3;            (* FC03 = read holding      *)
read_target_cfg.Node       := 1;

IF lp_toggle THEN
    read_local_cfg.ElementCnt := 5;         (* 0x210B..0x210F           *)
    read_target_cfg.Addr      := 16#210C;   (* AB subtracts 1 -> wire 0x210B *)
ELSE
    read_local_cfg.ElementCnt := 7;         (* 0x2100..0x2106           *)
    read_target_cfg.Addr      := 16#2101;   (* AB subtracts 1 -> wire 0x2100 *)
END_IF;

mb_read_status(IN        := poll_timer.Q AND poll_phase,
              LocalCfg  := read_local_cfg,
              TargetCfg := read_target_cfg,
              LocalAddr := read_data);

(* --- On success: unpack the block that was just read (raw values; scaling
       happens downstream in the historian: Hz x100, V x10, torque % x10,
       power kW x1000). --- *)
IF mb_read_status.Q AND NOT mb_read_status.Error THEN
    IF lp_toggle THEN
        vfd_torque    := read_data[1];      (* 0x210B  torque   % x10   *)
        vfd_motor_rpm := read_data[2];      (* 0x210C  motor rpm        *)
        vfd_power     := read_data[5];      (* 0x210F  power    kW x1000 *)
    ELSE
        vfd_fault_code  := read_data[1];    (* 0x2100  fault code (0=ok). NOTE:
                                               this is the whole word. Low byte =
                                               fault, high byte = warning. The
                                               byte-split was dropped (Micro800 ST
                                               AND/SHR need bit-string operands and
                                               read_data is UDINT). vfd_warn_code
                                               stays reserved (0) -- not decoded. *)
        vfd_status_word := read_data[2];    (* 0x2101  status word (bits) *)
        (* read_data[3] = 0x2102 keypad "F" echo: skipped (reads 0 in comms mode) *)
        vfd_frequency   := read_data[4];    (* 0x2103  output freq Hz x100 *)
        vfd_current     := read_data[5];    (* 0x2104  output amps A x100  *)
        vfd_dc_bus      := read_data[6];    (* 0x2105  DC bus      V x10   *)
        vfd_voltage     := read_data[7];    (* 0x2106  output volts V x10  *)
        IF vfd_fault_code > 0 THEN
            vfd_last_fault := vfd_fault_code; (* latch the trip cause *)
        END_IF;
    END_IF;
    vfd_comm_ok := TRUE;
END_IF;

IF mb_read_status.Error THEN
    vfd_comm_ok   := FALSE;
    vfd_err_count := vfd_err_count + 1;
END_IF;

(* --- Operator clear for the last-fault latch (Modbus coil 000024) --- *)
IF last_fault_clear THEN
    vfd_last_fault   := 0;
    last_fault_clear := FALSE;
END_IF;

(* ===================================================================== *)
(* REGISTER MAP (V2.0)   HR addr = CCW 4000xx as mapped in the .ccwmod    *)
(* 0x2100 fault   vfd_fault_code/400119   0x2100hi warn vfd_warn_code/400120 *)
(* 0x2101 status  vfd_status_word/400118  (cmd)    freqcmd vfd_freq_cmd/400121 *)
(* 0x2103 freq    vfd_frequency/400107    0x2104 amps   vfd_current/400108   *)
(* 0x2105 dcbus   vfd_dc_bus/400110       0x2106 outV   vfd_voltage/400109   *)
(* 0x210B torque  vfd_torque/400122       0x210C rpm    vfd_motor_rpm/400123 *)
(* 0x210F power   vfd_power/400124        (PLC) latch   vfd_last_fault/400125 *)
(* ===================================================================== *)

(* ===================================================================== *)
(* PHASE B -- VFD CONTROL (write path)   [UNCHANGED from V1.8]           *)
(* Writes alternate with reads on Channel 2 via poll_phase. The drive     *)
(* obeys only if P00.20=1 / P00.21=2. vfd_ctrl_enable=FALSE => read-only. *)
(* ===================================================================== *)

dir_fwd := _IO_EM_DI_00 AND NOT _IO_EM_DI_01;
dir_rev := _IO_EM_DI_01 AND NOT _IO_EM_DI_00;

IF _IO_EM_DI_05 THEN
    pe_latched := TRUE;        (* beam blocked -> latch the soft stop      *)
ELSIF _IO_EM_DI_04 THEN
    pe_latched := FALSE;       (* Start pressed (beam clear) -> rearm      *)
END_IF;

vfd_run_permit := _IO_EM_DO_02 AND e_stop_ok AND NOT pe_latched;

IF vfd_ctrl_enable AND vfd_run_permit AND dir_fwd THEN
    vfd_cmd_word := 18;        (* FWD + RUN *)
ELSIF vfd_ctrl_enable AND vfd_run_permit AND dir_rev THEN
    vfd_cmd_word := 34;        (* REV + RUN *)
ELSE
    vfd_cmd_word := 1;         (* STOP *)
END_IF;

IF vfd_freq_sp = 0 THEN
    vfd_freq_sp := 3000;       (* 30.00 Hz default *)
END_IF;

(* Frequency command (HR 400121) = the value the PLC writes to drive 0x2001.
   Always fresh, independent of the RS-485 read link, and is the true commanded
   Hz -- so the historian's freq-command-vs-output 1:1 check works. vfd_freq_sp
   is x100 (3000 = 30.00 Hz), same scale as vfd_freq_cmd. If Build flags a type
   mismatch here, vfd_freq_sp is not WORD -- declare a same-type intermediate or
   match the type; do NOT add ANY_TO_* (err 0124). *)
vfd_freq_cmd := vfd_freq_sp;

motor_running := vfd_run_permit AND (dir_fwd OR dir_rev);

write_local_cfg.Channel     := 2;
write_local_cfg.TriggerType := 0;
write_local_cfg.Cmd         := 16;         (* FC16 = write multiple    *)
write_local_cfg.ElementCnt  := 2;          (* cmd word + freq setpoint *)
write_target_cfg.Node := 1;
write_target_cfg.Addr := 16#2001;          (* AB subtracts 1 -> wire 0x2000 *)
write_cmd_data[1] := vfd_cmd_word;
write_cmd_data[2] := vfd_freq_sp;

mb_write_cmd(IN        := poll_timer.Q AND NOT poll_phase AND vfd_ctrl_enable,
             LocalCfg  := write_local_cfg,
             TargetCfg := write_target_cfg,
             LocalAddr := write_cmd_data);

IF mb_write_cmd.Error THEN
    vfd_err_count := vfd_err_count + 1;
END_IF;

END_PROGRAM
